LIN {X 0,Y 173.753,Z 484.675,A -85,B 0,C 180,E1 -23523.059,E2 -23523.059} C_VEL
LIN {X 0,Y 169.209,Z 473.205,A -85,B 0,C 180,E1 -23526.461,E2 -23526.461} C_VEL
LIN {X 0,Y 168.375,Z 468.327,A -85,B 0,C 180,E1 -23527.591,E2 -23527.591} C_VEL
LIN {X 0,Y 167.185,Z 457.036,A -85,B 0,C 180,E1 -23529.768,E2 -23529.768} C_VEL
LIN {X 0,Y 165.536,Z 447.869,A -85,B 0,C 180,E1 -23531.391,E2 -23531.391} C_VEL
LIN {X 0,Y 162.65,Z 440.385,A -85,B 0,C 180,E1 -23532.953,E2 -23532.953} C_VEL
LIN {X 0,Y 161.077,Z 436.839,A -85,B 0,C 180,E1 -23533.695,E2 -23533.695} C_VEL
LIN {X 0,Y 159.754,Z 433.864,A -85,B 0,C 180,E1 -23534.312,E2 -23534.312} C_VEL
LIN {X 0,Y 159.528,Z 432.773,A -85,B 0,C 180,E1 -23534.505,E2 -23534.505} C_VEL
LIN {X 0,Y 158.912,Z 429.909,A -85,B 0,C 180,E1 -23538.756,E2 -23538.756} C_VEL
LIN {X 0,Y 158.146,Z 426.115,A -85,B 0,C 180,E1 -23544.709,E2 -23544.709} C_VEL
LIN {X 0,Y 157.921,Z 424.301,A -85,B 0,C 180,E1 -23547.739,E2 -23547.739} C_VEL
LIN {X 0,Y 157.435,Z 421.293,A -85,B 0,C 180,E1 -23553.237,E2 -23553.237} C_VEL
LIN {X 0,Y 157.384,Z 420.882,A -85,B 0,C 180,E1 -23554.19,E2 -23554.19} C_VEL
LIN {X 0,Y 157.405,Z 420.883,A -85,B 0,C 180,E1 -23559.669,E2 -23559.669} C_VEL
LIN {X 0,Y 157.452,Z 420.881,A -85,B 0,C 180,E1 -23564.465,E2 -23564.465} C_VEL
LIN {X 0,Y 157.7,Z 420.846,A -85,B 0,C 180,E1 -23569.731,E2 -23569.731} C_VEL
LIN {X 0,Y 157.777,Z 420.836,A -85,B 0,C 180,E1 -23572.32,E2 -23572.32} C_VEL
LIN {X 0,Y 158.266,Z 420.771,A -85,B 0,C 180,E1 -23580,E2 -23580} C_VEL
LIN {X 0,Y 157.819,Z 420.787,A -85,B 0,C 180,E1 -23587.677,E2 -23587.677} C_VEL
LIN {X 0,Y 157.694,Z 420.835,A -85,B 0,C 180,E1 -23591.319,E2 -23591.319} C_VEL
LIN {X 0,Y 157.488,Z 420.862,A -85,B 0,C 180,E1 -23595.53,E2 -23595.53} C_VEL
LIN {X 0,Y 157.38,Z 420.844,A -85,B 0,C 180,E1 -23600.931,E2 -23600.931} C_VEL
LIN {X 0,Y 157.32,Z 420.888,A -85,B 0,C 180,E1 -23606.679,E2 -23606.679} C_VEL
LIN {X 0,Y 157.284,Z 420.858,A -85,B 0,C 180,E1 -23612.425,E2 -23612.425} C_VEL
LIN {X 0,Y 157.277,Z 420.888,A -85,B 0,C 180,E1 -23616.447,E2 -23616.447} C_VEL
LIN {X 0,Y 157.219,Z 420.881,A -85,B 0,C 180,E1 -23622.108,E2 -23622.108} C_VEL
LIN {X 0,Y 157.218,Z 420.901,A -85,B 0,C 180,E1 -23627.886,E2 -23627.886} C_VEL
LIN {X 0,Y 157.275,Z 420.879,A -85,B 0,C 180,E1 -23633.547,E2 -23633.547} C_VEL
LIN {X 0,Y 157.3,Z 420.889,A -85,B 0,C 180,E1 -23638.092,E2 -23638.092} C_VEL
LIN {X 0,Y 157.329,Z 420.894,A -85,B 0,C 180,E1 -23643.462,E2 -23643.462} C_VEL
LIN {X 0,Y 157.389,Z 421.075,A -85,B 0,C 180,E1 -23648.38,E2 -23648.38} C_VEL
LIN {X 0,Y 158.508,Z 423.935,A -85,B 0,C 180,E1 -23648.983,E2 -23648.983} C_VEL
LIN {X 0,Y 159.904,Z 425.81,A -85,B 0,C 180,E1 -23649.596,E2 -23649.596} C_VEL
LIN {X 0,Y 165.093,Z 435.684,A -85,B 0,C 180,E1 -23652.243,E2 -23652.243} C_VEL
LIN {X 0,Y 168.754,Z 444.416,A -85,B 0,C 180,E1 -23654.504,E2 -23654.504} C_VEL
LIN {X 0,Y 170.95,Z 453.105,A -85,B 0,C 180,E1 -23656.647,E2 -23656.647} C_VEL
LIN {X 0,Y 172.347,Z 463.912,A -85,B 0,C 180,E1 -23659.379,E2 -23659.379} C_VEL
LIN {X 0,Y 172.769,Z 470.682,A -85,B 0,C 180,E1 -23661.268,E2 -23661.268} C_VEL
LIN {X 0,Y 169.378,Z 481.319,A -85,B 0,C 180,E1 -23664.012,E2 -23664.012} C_VEL
LIN {X 0,Y 166.199,Z 490.266,A -85,B 0,C 180,E1 -23666.965,E2 -23666.965} C_VEL
LIN {X 0,Y 163.011,Z 498.684,A -85,B 0,C 180,E1 -23670.539,E2 -23670.539} C_VEL
LIN {X 0,Y 160.315,Z 505.722,A -85,B 0,C 180,E1 -23674.395,E2 -23674.395} C_VEL
LIN {X 0,Y 158.539,Z 510.345,A -85,B 0,C 180,E1 -23677.637,E2 -23677.637} C_VEL
LIN {X 0,Y 156.952,Z 514.644,A -85,B 0,C 180,E1 -23681.489,E2 -23681.489} C_VEL
LIN {X 0,Y 155.686,Z 518.09,A -85,B 0,C 180,E1 -23685.71,E2 -23685.71} C_VEL
LIN {X 0,Y 155.154,Z 519.7,A -85,B 0,C 180,E1 -23688.481,E2 -23688.481} C_VEL
LIN {X 0,Y 154.951,Z 520.827,A -85,B 0,C 180,E1 -23691.27,E2 -23691.27} C_VEL
LIN {X 0,Y 155.024,Z 521.64,A -85,B 0,C 180,E1 -23694.948,E2 -23694.948} C_VEL
LIN {X 0,Y 155.781,Z 521.51,A -85,B 0,C 180,E1 -23699.746,E2 -23699.746} C_VEL
LIN {X 0,Y 156.591,Z 520.823,A -85,B 0,C 180,E1 -23702.58,E2 -23702.58} C_VEL
LIN {X 0,Y 158.428,Z 518.701,A -85,B 0,C 180,E1 -23707.014,E2 -23707.014} C_VEL
LIN {X 0,Y 160.723,Z 515.657,A -85,B 0,C 180,E1 -23710.981,E2 -23710.981} C_VEL
LIN {X 0,Y 163.815,Z 511.176,A -85,B 0,C 180,E1 -23715.055,E2 -23715.055} C_VEL
LIN {X 0,Y 167.633,Z 505.239,A -85,B 0,C 180,E1 -23718.986,E2 -23718.986} C_VEL
LIN {X 0,Y 171.512,Z 498.72,A -85,B 0,C 180,E1 -23722.247,E2 -23722.247} C_VEL
LIN {X 0,Y 175.508,Z 491.246,A -85,B 0,C 180,E1 -23725.165,E2 -23725.165} C_VEL
LIN {X 0,Y 180.132,Z 481.611,A -85,B 0,C 180,E1 -23728.049,E2 -23728.049} C_VEL
LIN {X 0,Y 180.912,Z 479.34,A -85,B 0,C 180,E1 -23728.711,E2 -23728.711} C_VEL
LIN {X 0,Y 180.836,Z 471.499,A -85,B 0,C 180,E1 -23731.57,E2 -23731.57} C_VEL
LIN {X 0,Y 180.166,Z 465.408,A -85,B 0,C 180,E1 -23733.78,E2 -23733.78} C_VEL
LIN {X 0,Y 178.357,Z 457.69,A -85,B 0,C 180,E1 -23736.794,E2 -23736.794} C_VEL
LIN {X 0,Y 175.967,Z 451.426,A -85,B 0,C 180,E1 -23739.545,E2 -23739.545} C_VEL
LIN {X 0,Y 174.463,Z 447.925,A -85,B 0,C 180,E1 -23741.2,E2 -23741.2} C_VEL
LIN {X 0,Y 171.091,Z 441.961,A -85,B 0,C 180,E1 -23744.514,E2 -23744.514} C_VEL
LIN {X 0,Y 168.78,Z 438.136,A -85,B 0,C 180,E1 -23746.914,E2 -23746.914} C_VEL
LIN {X 0,Y 166.844,Z 434.787,A -85,B 0,C 180,E1 -23749.072,E2 -23749.072} C_VEL
LIN {X 0,Y 166.071,Z 433.805,A -85,B 0,C 180,E1 -23749.902,E2 -23749.902} C_VEL
LIN {X 0,Y 163.624,Z 430.698,A -85,B 0,C 180,E1 -23752.752,E2 -23752.752} C_VEL
LIN {X 0,Y 162.937,Z 429.155,A -85,B 0,C 180,E1 -23753.811,E2 -23753.811} C_VEL
LIN {X 0,Y 160.283,Z 427.137,A -85,B 0,C 180,E1 -23757.33,E2 -23757.33} C_VEL
LIN {X 0,Y 159.035,Z 424.704,A -85,B 0,C 180,E1 -23759.842,E2 -23759.842} C_VEL
LIN {X 0,Y 158.704,Z 423.885,A -85,B 0,C 180,E1 -23760.793,E2 -23760.793} C_VEL
LIN {X 0,Y 158.42,Z 424.419,A -85,B 0,C 180,E1 -23767.648,E2 -23767.648} C_VEL
LIN {X 0,Y 158.386,Z 425.205,A -85,B 0,C 180,E1 -23772.819,E2 -23772.819} C_VEL
LIN {X 0,Y 158.473,Z 426.363,A -85,B 0,C 180,E1 -23778.086,E2 -23778.086} C_VEL
LIN {X 0,Y 158.651,Z 427.629,A -85,B 0,C 180,E1 -23782.159,E2 -23782.159} C_VEL
LIN {X 0,Y 159.752,Z 430.657,A -85,B 0,C 180,E1 -23784.531,E2 -23784.531} C_VEL
LIN {X 0,Y 163.129,Z 435.032,A -85,B 0,C 180,E1 -23789.168,E2 -23789.168} C_VEL
LIN {X 0,Y 163.642,Z 435.727,A -85,B 0,C 180,E1 -23789.774,E2 -23789.774} C_VEL
LIN {X 0,Y 165.237,Z 439.58,A -85,B 0,C 180,E1 -23791.945,E2 -23791.945} C_VEL
LIN {X 0,Y 167.427,Z 442.4,A -85,B 0,C 180,E1 -23794.092,E2 -23794.092} C_VEL
LIN {X 0,Y 169.032,Z 446.242,A -85,B 0,C 180,E1 -23795.965,E2 -23795.965} C_VEL
LIN {X 0,Y 170.595,Z 448.842,A -85,B 0,C 180,E1 -23797.421,E2 -23797.421} C_VEL
LIN {X 0,Y 172.933,Z 453.744,A -85,B 0,C 180,E1 -23799.723,E2 -23799.723} C_VEL
LIN {X 0,Y 176.427,Z 462.831,A -85,B 0,C 180,E1 -23803.407,E2 -23803.407} C_VEL
LIN {X 0,Y 177.631,Z 467.087,A -85,B 0,C 180,E1 -23804.92,E2 -23804.92} C_VEL
LIN {X 0,Y 178.101,Z 473.747,A -85,B 0,C 180,E1 -23806.829,E2 -23806.829} C_VEL
LIN {X 0,Y 177.816,Z 483.644,A -85,B 0,C 180,E1 -23809.587,E2 -23809.587} C_VEL
LIN {X 0,Y 176.545,Z 493.509,A -85,B 0,C 180,E1 -23812.489,E2 -23812.489} C_VEL
LIN {X 0,Y 174.717,Z 501.481,A -85,B 0,C 180,E1 -23815.041,E2 -23815.041} C_VEL
LIN {X 0,Y 172.499,Z 508.067,A -85,B 0,C 180,E1 -23817.334,E2 -23817.334} C_VEL
LIN {X 0,Y 168.012,Z 516.355,A -85,B 0,C 180,E1 -23820.566,E2 -23820.566} C_VEL
LIN {X 0,Y 164.25,Z 523.057,A -85,B 0,C 180,E1 -23823.97,E2 -23823.97} C_VEL
LIN {X 0,Y 161.64,Z 527.705,A -85,B 0,C 180,E1 -23826.969,E2 -23826.969} C_VEL
LIN {X 0,Y 158.969,Z 532.18,A -85,B 0,C 180,E1 -23830.641,E2 -23830.641} C_VEL
LIN {X 0,Y 156.937,Z 535.616,A -85,B 0,C 180,E1 -23834.419,E2 -23834.419} C_VEL
LIN {X 0,Y 155.458,Z 538.718,A -85,B 0,C 180,E1 -23839.587,E2 -23839.587} C_VEL
LIN {X 0,Y 155.109,Z 539.685,A -85,B 0,C 180,E1 -23842.193,E2 -23842.193} C_VEL
LIN {X 0,Y 154.991,Z 540.343,A -85,B 0,C 180,E1 -23846.019,E2 -23846.019} C_VEL
LIN {X 0,Y 155.28,Z 540.125,A -85,B 0,C 180,E1 -23850.005,E2 -23850.005} C_VEL
LIN {X 0,Y 155.086,Z 538.698,A -85,B 0,C 180,E1 -23854.455,E2 -23854.455} C_VEL
LIN {X 0,Y 155.202,Z 536.785,A -85,B 0,C 180,E1 -23857.813,E2 -23857.813} C_VEL
LIN {X 0,Y 155.82,Z 533.633,A -85,B 0,C 180,E1 -23861.715,E2 -23861.715} C_VEL
LIN {X 0,Y 156.959,Z 529.391,A -85,B 0,C 180,E1 -23865.589,E2 -23865.589} C_VEL
LIN {X 0,Y 159.262,Z 522.952,A -85,B 0,C 180,E1 -23870.003,E2 -23870.003} C_VEL
LIN {X 0,Y 161.829,Z 515.818,A -85,B 0,C 180,E1 -23873.726,E2 -23873.726} C_VEL
LIN {X 0,Y 165.001,Z 507.05,A -85,B 0,C 180,E1 -23877.255,E2 -23877.255} C_VEL
LIN {X 0,Y 167.404,Z 499.95,A -85,B 0,C 180,E1 -23879.562,E2 -23879.562} C_VEL
LIN {X 0,Y 168.435,Z 489.968,A -85,B 0,C 180,E1 -23882.499,E2 -23882.499} C_VEL
LIN {X 0,Y 168.701,Z 478.718,A -85,B 0,C 180,E1 -23885.342,E2 -23885.342} C_VEL
LIN {X 0,Y 168.375,Z 468.327,A -85,B 0,C 180,E1 -23887.591,E2 -23887.591} C_VEL
LIN {X 0,Y 167.531,Z 463.422,A -85,B 0,C 180,E1 -23888.683,E2 -23888.683} C_VEL
LIN {X 0,Y 165.736,Z 458.883,A -85,B 0,C 180,E1 -23889.856,E2 -23889.856} C_VEL
LIN {X 0,Y 160.747,Z 450.349,A -85,B 0,C 180,E1 -23892.302,E2 -23892.302} C_VEL
LIN {X 0,Y 157.439,Z 444.408,A -85,B 0,C 180,E1 -23893.892,E2 -23893.892} C_VEL
LIN {X 0,Y 154.137,Z 436.914,A -85,B 0,C 180,E1 -23895.641,E2 -23895.641} C_VEL
LIN {X 0,Y 152.568,Z 433.873,A -85,B 0,C 180,E1 -23896.41,E2 -23896.41} C_VEL
LIN {X 0,Y 152.182,Z 432.293,A -85,B 0,C 180,E1 -23896.743,E2 -23896.743} C_VEL
LIN {X 0,Y 151.359,Z 428.42,A -85,B 0,C 180,E1 -23902.87,E2 -23902.87} C_VEL
LIN {X 0,Y 150.793,Z 424.852,A -85,B 0,C 180,E1 -23909.157,E2 -23909.157} C_VEL
LIN {X 0,Y 150.334,Z 421.76,A -85,B 0,C 180,E1 -23915.302,E2 -23915.302} C_VEL
LIN {X 0,Y 150.371,Z 421.761,A -85,B 0,C 180,E1 -23920.903,E2 -23920.903} C_VEL
LIN {X 0,Y 150.441,Z 421.754,A -85,B 0,C 180,E1 -23926.492,E2 -23926.492} C_VEL
LIN {X 0,Y 150.622,Z 421.728,A -85,B 0,C 180,E1 -23929.243,E2 -23929.243} C_VEL
LIN {X 0,Y 150.715,Z 421.715,A -85,B 0,C 180,E1 -23931.958,E2 -23931.958} C_VEL
LIN {X 0,Y 151.226,Z 421.648,A -85,B 0,C 180,E1 -23940,E2 -23940} C_VEL
LIN {X 0,Y 150.754,Z 421.667,A -85,B 0,C 180,E1 -23948.039,E2 -23948.039} C_VEL
LIN {X 0,Y 150.625,Z 421.716,A -85,B 0,C 180,E1 -23951.505,E2 -23951.505} C_VEL
LIN {X 0,Y 150.393,Z 421.741,A -85,B 0,C 180,E1 -23956.283,E2 -23956.283} C_VEL
LIN {X 0,Y 150.361,Z 421.716,A -85,B 0,C 180,E1 -23960.79,E2 -23960.79} C_VEL
LIN {X 0,Y 150.251,Z 421.77,A -85,B 0,C 180,E1 -23967.278,E2 -23967.278} C_VEL
LIN {X 0,Y 150.223,Z 421.736,A -85,B 0,C 180,E1 -23972.629,E2 -23972.629} C_VEL
LIN {X 0,Y 150.186,Z 421.775,A -85,B 0,C 180,E1 -23977.469,E2 -23977.469} C_VEL
LIN {X 0,Y 150.158,Z 421.766,A -85,B 0,C 180,E1 -23981.502,E2 -23981.502} C_VEL
LIN {X 0,Y 150.133,Z 421.764,A -85,B 0,C 180,E1 -23985.392,E2 -23985.392} C_VEL
LIN {X 0,Y 150.158,Z 421.78,A -85,B 0,C 180,E1 -23989.055,E2 -23989.055} C_VEL
LIN {X 0,Y 150.186,Z 421.758,A -85,B 0,C 180,E1 -23992.704,E2 -23992.704} C_VEL
LIN {X 0,Y 150.222,Z 421.775,A -85,B 0,C 180,E1 -23997.364,E2 -23997.364} C_VEL
LIN {X 0,Y 150.251,Z 421.776,A -85,B 0,C 180,E1 -24002.713,E2 -24002.713} C_VEL
LIN {X 0,Y 150.284,Z 421.83,A -85,B 0,C 180,E1 -24006.221,E2 -24006.221} C_VEL
LIN {X 0,Y 151.27,Z 424.573,A -85,B 0,C 180,E1 -24006.829,E2 -24006.829} C_VEL
LIN {X 0,Y 152.832,Z 426.794,A -85,B 0,C 180,E1 -24007.597,E2 -24007.597} C_VEL
LIN {X 0,Y 154.829,Z 430.108,A -85,B 0,C 180,E1 -24008.615,E2 -24008.615} C_VEL
LIN {X 0,Y 160.094,Z 440.601,A -85,B 0,C 180,E1 -24011.69,E2 -24011.69} C_VEL
LIN {X 0,Y 163.298,Z 449.135,A -85,B 0,C 180,E1 -24014.079,E2 -24014.079} C_VEL
LIN {X 0,Y 164.823,Z 455.727,A -85,B 0,C 180,E1 -24015.821,E2 -24015.821} C_VEL
LIN {X 0,Y 166.061,Z 467.475,A -85,B 0,C 180,E1 -24019.048,E2 -24019.048} C_VEL
LIN {X 0,Y 166.289,Z 471.524,A -85,B 0,C 180,E1 -24020.263,E2 -24020.263} C_VEL
LIN {X 0,Y 162.824,Z 482.07,A -85,B 0,C 180,E1 -24023.098,E2 -24023.098} C_VEL
LIN {X 0,Y 159.462,Z 491.064,A -85,B 0,C 180,E1 -24026.205,E2 -24026.205} C_VEL
LIN {X 0,Y 156.081,Z 499.578,A -85,B 0,C 180,E1 -24029.995,E2 -24029.995} C_VEL
LIN {X 0,Y 153.342,Z 506.408,A -85,B 0,C 180,E1 -24033.937,E2 -24033.937} C_VEL
LIN {X 0,Y 151.177,Z 511.81,A -85,B 0,C 180,E1 -24038.012,E2 -24038.012} C_VEL
LIN {X 0,Y 149.56,Z 515.99,A -85,B 0,C 180,E1 -24042.202,E2 -24042.202} C_VEL
LIN {X 0,Y 148.413,Z 519.07,A -85,B 0,C 180,E1 -24046.501,E2 -24046.501} C_VEL
LIN {X 0,Y 147.979,Z 520.528,A -85,B 0,C 180,E1 -24049.412,E2 -24049.412} C_VEL
LIN {X 0,Y 147.827,Z 521.555,A -85,B 0,C 180,E1 -24052.348,E2 -24052.348} C_VEL
LIN {X 0,Y 147.975,Z 522.1,A -85,B 0,C 180,E1 -24055.525,E2 -24055.525} C_VEL
LIN {X 0,Y 148.359,Z 522.166,A -85,B 0,C 180,E1 -24058.269,E2 -24058.269} C_VEL
LIN {X 0,Y 149.353,Z 521.577,A -85,B 0,C 180,E1 -24062.112,E2 -24062.112} C_VEL
LIN {X 0,Y 151.319,Z 519.586,A -85,B 0,C 180,E1 -24067.134,E2 -24067.134} C_VEL
LIN {X 0,Y 153.807,Z 516.595,A -85,B 0,C 180,E1 -24071.487,E2 -24071.487} C_VEL
LIN {X 0,Y 157.041,Z 512.303,A -85,B 0,C 180,E1 -24075.72,E2 -24075.72} C_VEL
LIN {X 0,Y 161.031,Z 506.509,A -85,B 0,C 180,E1 -24079.818,E2 -24079.818} C_VEL
LIN {X 0,Y 165.708,Z 499.132,A -85,B 0,C 180,E1 -24083.68,E2 -24083.68} C_VEL
LIN {X 0,Y 169.998,Z 491.579,A -85,B 0,C 180,E1 -24086.686,E2 -24086.686} C_VEL
LIN {X 0,Y 174.948,Z 481.709,A -85,B 0,C 180,E1 -24089.69,E2 -24089.69} C_VEL
LIN {X 0,Y 175.119,Z 474.619,A -85,B 0,C 180,E1 -24092.476,E2 -24092.476} C_VEL
LIN {X 0,Y 174.394,Z 466.778,A -85,B 0,C 180,E1 -24095.602,E2 -24095.602} C_VEL
LIN {X 0,Y 172.779,Z 460.047,A -85,B 0,C 180,E1 -24098.526,E2 -24098.526} C_VEL
LIN {X 0,Y 170.226,Z 453.171,A -85,B 0,C 180,E1 -24101.961,E2 -24101.961} C_VEL
LIN {X 0,Y 166.794,Z 446.29,A -85,B 0,C 180,E1 -24106.041,E2 -24106.041} C_VEL
LIN {X 0,Y 163.603,Z 440.467,A -85,B 0,C 180,E1 -24110.106,E2 -24110.106} C_VEL
LIN {X 0,Y 161.169,Z 437.172,A -85,B 0,C 180,E1 -24113.31,E2 -24113.31} C_VEL
LIN {X 0,Y 160.584,Z 435.793,A -85,B 0,C 180,E1 -24114.356,E2 -24114.356} C_VEL
LIN {X 0,Y 158.165,Z 433.6,A -85,B 0,C 180,E1 -24118.09,E2 -24118.09} C_VEL
LIN {X 0,Y 157.097,Z 430.867,A -85,B 0,C 180,E1 -24120.961,E2 -24120.961} C_VEL
LIN {X 0,Y 154.798,Z 430.545,A -85,B 0,C 180,E1 -24127.828,E2 -24127.828} C_VEL
LIN {X 0,Y 154.562,Z 431.276,A -85,B 0,C 180,E1 -24133.141,E2 -24133.141} C_VEL
LIN {X 0,Y 156.749,Z 434.093,A -85,B 0,C 180,E1 -24141.208,E2 -24141.208} C_VEL
LIN {X 0,Y 158.112,Z 437.966,A -85,B 0,C 180,E1 -24144.628,E2 -24144.628} C_VEL
LIN {X 0,Y 160.988,Z 442.005,A -85,B 0,C 180,E1 -24148.94,E2 -24148.94} C_VEL
LIN {X 0,Y 162.573,Z 446.035,A -85,B 0,C 180,E1 -24151.438,E2 -24151.438} C_VEL
LIN {X 0,Y 163.813,Z 447.698,A -85,B 0,C 180,E1 -24152.812,E2 -24152.812} C_VEL
LIN {X 0,Y 166.556,Z 453.649,A -85,B 0,C 180,E1 -24156.21,E2 -24156.21} C_VEL
LIN {X 0,Y 169.063,Z 459.815,A -85,B 0,C 180,E1 -24159.236,E2 -24159.236} C_VEL
LIN {X 0,Y 171.629,Z 467.332,A -85,B 0,C 180,E1 -24162.525,E2 -24162.525} C_VEL
LIN {X 0,Y 172.625,Z 472.125,A -85,B 0,C 180,E1 -24164.297,E2 -24164.297} C_VEL
LIN {X 0,Y 172.583,Z 480.365,A -85,B 0,C 180,E1 -24166.786,E2 -24166.786} C_VEL
LIN {X 0,Y 171.457,Z 490.287,A -85,B 0,C 180,E1 -24169.798,E2 -24169.798} C_VEL
LIN {X 0,Y 169.619,Z 499.083,A -85,B 0,C 180,E1 -24172.676,E2 -24172.676} C_VEL
LIN {X 0,Y 167.17,Z 506.719,A -85,B 0,C 180,E1 -24175.427,E2 -24175.427} C_VEL
LIN {X 0,Y 164.15,Z 512.526,A -85,B 0,C 180,E1 -24177.65,E2 -24177.65} C_VEL
LIN {X 0,Y 159.751,Z 519.896,A -85,B 0,C 180,E1 -24181.064,E2 -24181.064} C_VEL
LIN {X 0,Y 156.249,Z 525.875,A -85,B 0,C 180,E1 -24184.709,E2 -24184.709} C_VEL
LIN {X 0,Y 153.122,Z 530.645,A -85,B 0,C 180,E1 -24188.464,E2 -24188.464} C_VEL
LIN {X 0,Y 150.724,Z 534.341,A -85,B 0,C 180,E1 -24192.363,E2 -24192.363} C_VEL
LIN {X 0,Y 149.115,Z 537.064,A -85,B 0,C 180,E1 -24196.375,E2 -24196.375} C_VEL
LIN {X 0,Y 148.463,Z 538.386,A -85,B 0,C 180,E1 -24199.09,E2 -24199.09} C_VEL
LIN {X 0,Y 148.042,Z 539.306,A -85,B 0,C 180,E1 -24201.818,E2 -24201.818} C_VEL
LIN {X 0,Y 147.915,Z 539.947,A -85,B 0,C 180,E1 -24206.193,E2 -24206.193} C_VEL
LIN {X 0,Y 148.192,Z 539.65,A -85,B 0,C 180,E1 -24210.005,E2 -24210.005} C_VEL
LIN {X 0,Y 147.996,Z 538.335,A -85,B 0,C 180,E1 -24214.251,E2 -24214.251} C_VEL
LIN {X 0,Y 148.309,Z 535.251,A -85,B 0,C 180,E1 -24219.552,E2 -24219.552} C_VEL
LIN {X 0,Y 149.173,Z 531.684,A -85,B 0,C 180,E1 -24223.63,E2 -24223.63} C_VEL
LIN {X 0,Y 150.752,Z 526.998,A -85,B 0,C 180,E1 -24227.645,E2 -24227.645} C_VEL
LIN {X 0,Y 153.39,Z 519.918,A -85,B 0,C 180,E1 -24232.215,E2 -24232.215} C_VEL
LIN {X 0,Y 156.109,Z 512.72,A -85,B 0,C 180,E1 -24235.789,E2 -24235.789} C_VEL
LIN {X 0,Y 159.296,Z 504.366,A -85,B 0,C 180,E1 -24239.038,E2 -24239.038} C_VEL
LIN {X 0,Y 160.802,Z 499.788,A -85,B 0,C 180,E1 -24240.541,E2 -24240.541} C_VEL
LIN {X 0,Y 161.84,Z 489.809,A -85,B 0,C 180,E1 -24243.625,E2 -24243.625} C_VEL
LIN {X 0,Y 162.213,Z 480.188,A -85,B 0,C 180,E1 -24246.183,E2 -24246.183} C_VEL
LIN {X 0,Y 162.028,Z 469.456,A -85,B 0,C 180,E1 -24248.67,E2 -24248.67} C_VEL
LIN {X 0,Y 160.969,Z 457.998,A -85,B 0,C 180,E1 -24251.042,E2 -24251.042} C_VEL
LIN {X 0,Y 159.68,Z 450.554,A -85,B 0,C 180,E1 -24252.504,E2 -24252.504} C_VEL
LIN {X 0,Y 157.439,Z 444.408,A -85,B 0,C 180,E1 -24253.892,E2 -24253.892} C_VEL
LIN {X 0,Y 155.429,Z 441.819,A -85,B 0,C 180,E1 -24254.754,E2 -24254.754} C_VEL
LIN {X 0,Y 146.78,Z 436.045,A -85,B 0,C 180,E1 -24258.088,E2 -24258.088} C_VEL
LIN {X 0,Y 145.32,Z 433.745,A -85,B 0,C 180,E1 -24258.807,E2 -24258.807} C_VEL
LIN {X 0,Y 145.124,Z 433.196,A -85,B 0,C 180,E1 -24258.926,E2 -24258.926} C_VEL
LIN {X 0,Y 144.775,Z 431.726,A -85,B 0,C 180,E1 -24259.226,E2 -24259.226} C_VEL
LIN {X 0,Y 144.051,Z 427.842,A -85,B 0,C 180,E1 -24266.045,E2 -24266.045} C_VEL
LIN {X 0,Y 143.584,Z 424.839,A -85,B 0,C 180,E1 -24271.778,E2 -24271.778} C_VEL
LIN {X 0,Y 143.246,Z 422.643,A -85,B 0,C 180,E1 -24276.507,E2 -24276.507} C_VEL
LIN {X 0,Y 143.318,Z 422.639,A -85,B 0,C 180,E1 -24279.924,E2 -24279.924} C_VEL
LIN {X 0,Y 143.364,Z 422.634,A -85,B 0,C 180,E1 -24285.811,E2 -24285.811} C_VEL
LIN {X 0,Y 143.548,Z 422.611,A -85,B 0,C 180,E1 -24288.706,E2 -24288.706} C_VEL
LIN {X 0,Y 143.636,Z 422.597,A -85,B 0,C 180,E1 -24291.559,E2 -24291.559} C_VEL
LIN {X 0,Y 144.185,Z 422.525,A -85,B 0,C 180,E1 -24300,E2 -24300} C_VEL
LIN {X 0,Y 143.675,Z 422.55,A -85,B 0,C 180,E1 -24308.438,E2 -24308.438} C_VEL
LIN {X 0,Y 143.559,Z 422.597,A -85,B 0,C 180,E1 -24311.711,E2 -24311.711} C_VEL
LIN {X 0,Y 143.327,Z 422.611,A -85,B 0,C 180,E1 -24317.11,E2 -24317.11} C_VEL
LIN {X 0,Y 143.287,Z 422.598,A -85,B 0,C 180,E1 -24321.252,E2 -24321.252} C_VEL
LIN {X 0,Y 143.198,Z 422.645,A -85,B 0,C 180,E1 -24327.933,E2 -24327.933} C_VEL
LIN {X 0,Y 143.152,Z 422.617,A -85,B 0,C 180,E1 -24333.417,E2 -24333.417} C_VEL
LIN {X 0,Y 143.071,Z 422.661,A -85,B 0,C 180,E1 -24339.687,E2 -24339.687} C_VEL
LIN {X 0,Y 143.045,Z 422.638,A -85,B 0,C 180,E1 -24343.459,E2 -24343.459} C_VEL
LIN {X 0,Y 143.073,Z 422.661,A -85,B 0,C 180,E1 -24347.462,E2 -24347.462} C_VEL
LIN {X 0,Y 143.084,Z 422.643,A -85,B 0,C 180,E1 -24351.803,E2 -24351.803} C_VEL
LIN {X 0,Y 143.189,Z 422.651,A -85,B 0,C 180,E1 -24357.317,E2 -24357.317} C_VEL
LIN {X 0,Y 143.189,Z 422.655,A -85,B 0,C 180,E1 -24363.78,E2 -24363.78} C_VEL
LIN {X 0,Y 144.206,Z 425.52,A -85,B 0,C 180,E1 -24364.488,E2 -24364.488} C_VEL
LIN {X 0,Y 145.853,Z 427.689,A -85,B 0,C 180,E1 -24365.372,E2 -24365.372} C_VEL
LIN {X 0,Y 151.079,Z 437.022,A -85,B 0,C 180,E1 -24368.493,E2 -24368.493} C_VEL
LIN {X 0,Y 155.548,Z 446.838,A -85,B 0,C 180,E1 -24371.591,E2 -24371.591} C_VEL
LIN {X 0,Y 157.903,Z 454.279,A -85,B 0,C 180,E1 -24373.823,E2 -24373.823} C_VEL
LIN {X 0,Y 158.998,Z 461.758,A -85,B 0,C 180,E1 -24375.926,E2 -24375.926} C_VEL
LIN {X 0,Y 159.708,Z 470.646,A -85,B 0,C 180,E1 -24378.606,E2 -24378.606} C_VEL
LIN {X 0,Y 159.792,Z 472.598,A -85,B 0,C 180,E1 -24379.238,E2 -24379.238} C_VEL
LIN {X 0,Y 156.871,Z 481.215,A -85,B 0,C 180,E1 -24381.623,E2 -24381.623} C_VEL
LIN {X 0,Y 153.398,Z 490.265,A -85,B 0,C 180,E1 -24384.738,E2 -24384.738} C_VEL
LIN {X 0,Y 150.358,Z 497.708,A -85,B 0,C 180,E1 -24387.986,E2 -24387.986} C_VEL
LIN {X 0,Y 147.639,Z 504.135,A -85,B 0,C 180,E1 -24391.512,E2 -24391.512} C_VEL
LIN {X 0,Y 145.187,Z 509.901,A -85,B 0,C 180,E1 -24395.55,E2 -24395.55} C_VEL
LIN {X 0,Y 142.994,Z 515.26,A -85,B 0,C 180,E1 -24400.587,E2 -24400.587} C_VEL
LIN {X 0,Y 141.799,Z 518.208,A -85,B 0,C 180,E1 -24404.342,E2 -24404.342} C_VEL
LIN {X 0,Y 140.962,Z 520.627,A -85,B 0,C 180,E1 -24408.686,E2 -24408.686} C_VEL
LIN {X 0,Y 140.761,Z 522.186,A -85,B 0,C 180,E1 -24413.536,E2 -24413.536} C_VEL
LIN {X 0,Y 141.004,Z 522.598,A -85,B 0,C 180,E1 -24416.646,E2 -24416.646} C_VEL
LIN {X 0,Y 141.577,Z 522.563,A -85,B 0,C 180,E1 -24419.756,E2 -24419.756} C_VEL
LIN {X 0,Y 142.497,Z 521.976,A -85,B 0,C 180,E1 -24423.024,E2 -24423.024} C_VEL
LIN {X 0,Y 143.586,Z 521.025,A -85,B 0,C 180,E1 -24425.962,E2 -24425.962} C_VEL
LIN {X 0,Y 145.2,Z 519.384,A -85,B 0,C 180,E1 -24429.247,E2 -24429.247} C_VEL
LIN {X 0,Y 147.965,Z 516.26,A -85,B 0,C 180,E1 -24433.52,E2 -24433.52} C_VEL
LIN {X 0,Y 151.566,Z 511.701,A -85,B 0,C 180,E1 -24437.885,E2 -24437.885} C_VEL
LIN {X 0,Y 156.011,Z 505.695,A -85,B 0,C 180,E1 -24442.021,E2 -24442.021} C_VEL
LIN {X 0,Y 161.103,Z 497.863,A -85,B 0,C 180,E1 -24445.972,E2 -24445.972} C_VEL
LIN {X 0,Y 165.886,Z 489.7,A -85,B 0,C 180,E1 -24449.068,E2 -24449.068} C_VEL
LIN {X 0,Y 169.002,Z 483.889,A -85,B 0,C 180,E1 -24450.832,E2 -24450.832} C_VEL
LIN {X 0,Y 169.424,Z 477.503,A -85,B 0,C 180,E1 -24453.517,E2 -24453.517} C_VEL
LIN {X 0,Y 169.169,Z 471.632,A -85,B 0,C 180,E1 -24456.046,E2 -24456.046} C_VEL
LIN {X 0,Y 167.972,Z 464.902,A -85,B 0,C 180,E1 -24459.167,E2 -24459.167} C_VEL
LIN {X 0,Y 165.835,Z 458.262,A -85,B 0,C 180,E1 -24462.743,E2 -24462.743} C_VEL
LIN {X 0,Y 163.34,Z 452.656,A -85,B 0,C 180,E1 -24466.311,E2 -24466.311} C_VEL
LIN {X 0,Y 160.141,Z 446.233,A -85,B 0,C 180,E1 -24471.164,E2 -24471.164} C_VEL
LIN {X 0,Y 158.515,Z 443.876,A -85,B 0,C 180,E1 -24473.636,E2 -24473.636} C_VEL
LIN {X 0,Y 157.95,Z 442.293,A -85,B 0,C 180,E1 -24474.895,E2 -24474.895} C_VEL
LIN {X 0,Y 156.433,Z 440.982,A -85,B 0,C 180,E1 -24477.425,E2 -24477.425} C_VEL
LIN {X 0,Y 155.059,Z 437.806,A -85,B 0,C 180,E1 -24481.299,E2 -24481.299} C_VEL
LIN {X 0,Y 152.914,Z 437.537,A -85,B 0,C 180,E1 -24489.257,E2 -24489.257} C_VEL
LIN {X 0,Y 153.09,Z 438.741,A -85,B 0,C 180,E1 -24495.137,E2 -24495.137} C_VEL
LIN {X 0,Y 154.688,Z 440.97,A -85,B 0,C 180,E1 -24500.791,E2 -24500.791} C_VEL
LIN {X 0,Y 155.719,Z 444.389,A -85,B 0,C 180,E1 -24503.966,E2 -24503.966} C_VEL
LIN {X 0,Y 157.937,Z 447.777,A -85,B 0,C 180,E1 -24507.855,E2 -24507.855} C_VEL
LIN {X 0,Y 159.304,Z 451.768,A -85,B 0,C 180,E1 -24510.488,E2 -24510.488} C_VEL
LIN {X 0,Y 160.658,Z 454.19,A -85,B 0,C 180,E1 -24512.404,E2 -24512.404} C_VEL
LIN {X 0,Y 163.188,Z 460.792,A -85,B 0,C 180,E1 -24516.235,E2 -24516.235} C_VEL
LIN {X 0,Y 165.458,Z 467.333,A -85,B 0,C 180,E1 -24519.579,E2 -24519.579} C_VEL
LIN {X 0,Y 167.088,Z 473.304,A -85,B 0,C 180,E1 -24522.298,E2 -24522.298} C_VEL
LIN {X 0,Y 167.396,Z 477.452,A -85,B 0,C 180,E1 -24523.812,E2 -24523.812} C_VEL
LIN {X 0,Y 166.698,Z 485.785,A -85,B 0,C 180,E1 -24526.486,E2 -24526.486} C_VEL
LIN {X 0,Y 165.033,Z 494.869,A -85,B 0,C 180,E1 -24529.509,E2 -24529.509} C_VEL
LIN {X 0,Y 162.456,Z 503.778,A -85,B 0,C 180,E1 -24532.731,E2 -24532.731} C_VEL
LIN {X 0,Y 160.638,Z 508.439,A -85,B 0,C 180,E1 -24534.578,E2 -24534.578} C_VEL
LIN {X 0,Y 155.772,Z 516.494,A -85,B 0,C 180,E1 -24537.992,E2 -24537.992} C_VEL
LIN {X 0,Y 152.189,Z 522.016,A -85,B 0,C 180,E1 -24541.003,E2 -24541.003} C_VEL
LIN {X 0,Y 148.657,Z 527.47,A -85,B 0,C 180,E1 -24544.825,E2 -24544.825} C_VEL
LIN {X 0,Y 145.59,Z 531.788,A -85,B 0,C 180,E1 -24548.78,E2 -24548.78} C_VEL
LIN {X 0,Y 143.23,Z 535.088,A -85,B 0,C 180,E1 -24552.884,E2 -24552.884} C_VEL
LIN {X 0,Y 141.454,Z 538.057,A -85,B 0,C 180,E1 -24558.543,E2 -24558.543} C_VEL
LIN {X 0,Y 140.842,Z 539.387,A -85,B 0,C 180,E1 -24564.278,E2 -24564.278} C_VEL
LIN {X 0,Y 140.864,Z 539.471,A -85,B 0,C 180,E1 -24567.146,E2 -24567.146} C_VEL
LIN {X 0,Y 141.105,Z 539.171,A -85,B 0,C 180,E1 -24570.005,E2 -24570.005} C_VEL
LIN {X 0,Y 140.925,Z 537.929,A -85,B 0,C 180,E1 -24574.117,E2 -24574.117} C_VEL
LIN {X 0,Y 141.3,Z 534.615,A -85,B 0,C 180,E1 -24580.031,E2 -24580.031} C_VEL
LIN {X 0,Y 142.24,Z 530.977,A -85,B 0,C 180,E1 -24584.308,E2 -24584.308} C_VEL
LIN {X 0,Y 143.959,Z 526.217,A -85,B 0,C 180,E1 -24588.507,E2 -24588.507} C_VEL
LIN {X 0,Y 146.823,Z 519.058,A -85,B 0,C 180,E1 -24593.265,E2 -24593.265} C_VEL
LIN {X 0,Y 149.962,Z 511.09,A -85,B 0,C 180,E1 -24597.264,E2 -24597.264} C_VEL
LIN {X 0,Y 153.745,Z 501.447,A -85,B 0,C 180,E1 -24600.953,E2 -24600.953} C_VEL
LIN {X 0,Y 155.112,Z 492.417,A -85,B 0,C 180,E1 -24603.972,E2 -24603.972} C_VEL
LIN {X 0,Y 155.741,Z 481.499,A -85,B 0,C 180,E1 -24607.131,E2 -24607.131} C_VEL
LIN {X 0,Y 155.736,Z 470.304,A -85,B 0,C 180,E1 -24609.899,E2 -24609.899} C_VEL
LIN {X 0,Y 154.87,Z 459.374,A -85,B 0,C 180,E1 -24612.319,E2 -24612.319} C_VEL
LIN {X 0,Y 153.942,Z 453.583,A -85,B 0,C 180,E1 -24613.551,E2 -24613.551} C_VEL
LIN {X 0,Y 150.558,Z 444.438,A -85,B 0,C 180,E1 -24615.869,E2 -24615.869} C_VEL
LIN {X 0,Y 146.799,Z 436.365,A -85,B 0,C 180,E1 -24618.029,E2 -24618.029} C_VEL
LIN {X 0,Y 145.124,Z 433.196,A -85,B 0,C 180,E1 -24618.926,E2 -24618.926} C_VEL
LIN {X 0,Y 144.246,Z 431.755,A -85,B 0,C 180,E1 -24619.567,E2 -24619.567} C_VEL
LIN {X 0,Y 139.809,Z 429.739,A -85,B 0,C 180,E1 -24623.988,E2 -24623.988} C_VEL
LIN {X 0,Y 137.652,Z 428.46,A -85,B 0,C 180,E1 -24627.481,E2 -24627.481} C_VEL
LIN {X 0,Y 136.644,Z 426.536,A -85,B 0,C 180,E1 -24631.067,E2 -24631.067} C_VEL
LIN {X 0,Y 136.268,Z 423.809,A -85,B 0,C 180,E1 -24637.116,E2 -24637.116} C_VEL
LIN {X 0,Y 136.256,Z 423.517,A -85,B 0,C 180,E1 -24638.835,E2 -24638.835} C_VEL
LIN {X 0,Y 136.274,Z 423.518,A -85,B 0,C 180,E1 -24645.056,E2 -24645.056} C_VEL
LIN {X 0,Y 136.442,Z 423.497,A -85,B 0,C 180,E1 -24648.167,E2 -24648.167} C_VEL
LIN {X 0,Y 136.562,Z 423.479,A -85,B 0,C 180,E1 -24651.118,E2 -24651.118} C_VEL
LIN {X 0,Y 137.142,Z 423.402,A -85,B 0,C 180,E1 -24660,E2 -24660} C_VEL
LIN {X 0,Y 136.602,Z 423.434,A -85,B 0,C 180,E1 -24668.879,E2 -24668.879} C_VEL
LIN {X 0,Y 136.502,Z 423.477,A -85,B 0,C 180,E1 -24671.953,E2 -24671.953} C_VEL
LIN {X 0,Y 136.262,Z 423.479,A -85,B 0,C 180,E1 -24678.027,E2 -24678.027} C_VEL
LIN {X 0,Y 136.208,Z 423.481,A -85,B 0,C 180,E1 -24681.746,E2 -24681.746} C_VEL
LIN {X 0,Y 136.109,Z 423.524,A -85,B 0,C 180,E1 -24688.612,E2 -24688.612} C_VEL
LIN {X 0,Y 136.052,Z 423.508,A -85,B 0,C 180,E1 -24694.626,E2 -24694.626} C_VEL
LIN {X 0,Y 136.042,Z 423.538,A -85,B 0,C 180,E1 -24699.196,E2 -24699.196} C_VEL
LIN {X 0,Y 135.99,Z 423.515,A -85,B 0,C 180,E1 -24703.647,E2 -24703.647} C_VEL
LIN {X 0,Y 136.036,Z 423.54,A -85,B 0,C 180,E1 -24707.802,E2 -24707.802} C_VEL
LIN {X 0,Y 136.034,Z 423.521,A -85,B 0,C 180,E1 -24711.68,E2 -24711.68} C_VEL
LIN {X 0,Y 136.092,Z 423.534,A -85,B 0,C 180,E1 -24715.717,E2 -24715.717} C_VEL
LIN {X 0,Y 136.104,Z 423.532,A -85,B 0,C 180,E1 -24721.046,E2 -24721.046} C_VEL
LIN {X 0,Y 137.029,Z 426.189,A -85,B 0,C 180,E1 -24721.771,E2 -24721.771} C_VEL
LIN {X 0,Y 138.888,Z 428.715,A -85,B 0,C 180,E1 -24722.903,E2 -24722.903} C_VEL
LIN {X 0,Y 140.841,Z 432.005,A -85,B 0,C 180,E1 -24724.15,E2 -24724.15} C_VEL
LIN {X 0,Y 146.437,Z 442.379,A -85,B 0,C 180,E1 -24727.965,E2 -24727.965} C_VEL
LIN {X 0,Y 150.385,Z 451.906,A -85,B 0,C 180,E1 -24731.211,E2 -24731.211} C_VEL
LIN {X 0,Y 151.978,Z 457.537,A -85,B 0,C 180,E1 -24733.033,E2 -24733.033} C_VEL
LIN {X 0,Y 152.775,Z 464.096,A -85,B 0,C 180,E1 -24735.026,E2 -24735.026} C_VEL
LIN {X 0,Y 153.285,Z 472.924,A -85,B 0,C 180,E1 -24737.891,E2 -24737.891} C_VEL
LIN {X 0,Y 153.159,Z 474.532,A -85,B 0,C 180,E1 -24738.394,E2 -24738.394} C_VEL
LIN {X 0,Y 149.193,Z 485.07,A -85,B 0,C 180,E1 -24741.587,E2 -24741.587} C_VEL
LIN {X 0,Y 145.486,Z 494.115,A -85,B 0,C 180,E1 -24745.145,E2 -24745.145} C_VEL
LIN {X 0,Y 141.869,Z 502.211,A -85,B 0,C 180,E1 -24749.285,E2 -24749.285} C_VEL
LIN {X 0,Y 139.432,Z 507.698,A -85,B 0,C 180,E1 -24752.884,E2 -24752.884} C_VEL
LIN {X 0,Y 137.107,Z 512.995,A -85,B 0,C 180,E1 -24757.357,E2 -24757.357} C_VEL
LIN {X 0,Y 135.344,Z 517.105,A -85,B 0,C 180,E1 -24761.982,E2 -24761.982} C_VEL
LIN {X 0,Y 134.456,Z 519.239,A -85,B 0,C 180,E1 -24765.144,E2 -24765.144} C_VEL
LIN {X 0,Y 133.842,Z 521.183,A -85,B 0,C 180,E1 -24769.061,E2 -24769.061} C_VEL
LIN {X 0,Y 133.746,Z 522.805,A -85,B 0,C 180,E1 -24774.852,E2 -24774.852} C_VEL
LIN {X 0,Y 134.125,Z 523.086,A -85,B 0,C 180,E1 -24778.13,E2 -24778.13} C_VEL
LIN {X 0,Y 135.714,Z 522.37,A -85,B 0,C 180,E1 -24784.049,E2 -24784.049} C_VEL
LIN {X 0,Y 137.272,Z 521.072,A -85,B 0,C 180,E1 -24787.898,E2 -24787.898} C_VEL
LIN {X 0,Y 140,Z 518.386,A -85,B 0,C 180,E1 -24792.655,E2 -24792.655} C_VEL
LIN {X 0,Y 143.565,Z 514.464,A -85,B 0,C 180,E1 -24797.239,E2 -24797.239} C_VEL
LIN {X 0,Y 148.244,Z 508.715,A -85,B 0,C 180,E1 -24801.953,E2 -24801.953} C_VEL
LIN {X 0,Y 152.997,Z 502.238,A -85,B 0,C 180,E1 -24805.765,E2 -24805.765} C_VEL
LIN {X 0,Y 157.79,Z 494.982,A -85,B 0,C 180,E1 -24809.015,E2 -24809.015} C_VEL
LIN {X 0,Y 162.564,Z 486.928,A -85,B 0,C 180,E1 -24811.803,E2 -24811.803} C_VEL
LIN {X 0,Y 163.316,Z 485.147,A -85,B 0,C 180,E1 -24812.445,E2 -24812.445} C_VEL
LIN {X 0,Y 163.787,Z 479.083,A -85,B 0,C 180,E1 -24815.207,E2 -24815.207} C_VEL
LIN {X 0,Y 163.568,Z 473.394,A -85,B 0,C 180,E1 -24817.916,E2 -24817.916} C_VEL
LIN {X 0,Y 162.782,Z 468.547,A -85,B 0,C 180,E1 -24820.452,E2 -24820.452} C_VEL
LIN {X 0,Y 161.006,Z 462.576,A -85,B 0,C 180,E1 -24824.008,E2 -24824.008} C_VEL
LIN {X 0,Y 159.225,Z 457.84,A -85,B 0,C 180,E1 -24827.25,E2 -24827.25} C_VEL
LIN {X 0,Y 156.498,Z 451.866,A -85,B 0,C 180,E1 -24832.258,E2 -24832.258} C_VEL
LIN {X 0,Y 155.237,Z 449.394,A -85,B 0,C 180,E1 -24834.805,E2 -24834.805} C_VEL
LIN {X 0,Y 152.331,Z 444.337,A -85,B 0,C 180,E1 -24842.645,E2 -24842.645} C_VEL
LIN {X 0,Y 150.961,Z 444.233,A -85,B 0,C 180,E1 -24848.029,E2 -24848.029} C_VEL
LIN {X 0,Y 150.791,Z 445.086,A -85,B 0,C 180,E1 -24853.476,E2 -24853.476} C_VEL
LIN {X 0,Y 151.854,Z 446.84,A -85,B 0,C 180,E1 -24858.903,E2 -24858.903} C_VEL
LIN {X 0,Y 152.228,Z 447.642,A -85,B 0,C 180,E1 -24860.259,E2 -24860.259} C_VEL
LIN {X 0,Y 153.411,Z 451.635,A -85,B 0,C 180,E1 -24864.35,E2 -24864.35} C_VEL
LIN {X 0,Y 154.75,Z 453.809,A -85,B 0,C 180,E1 -24867.011,E2 -24867.011} C_VEL
LIN {X 0,Y 155.906,Z 457.61,A -85,B 0,C 180,E1 -24869.727,E2 -24869.727} C_VEL
LIN {X 0,Y 157.082,Z 460.183,A -85,B 0,C 180,E1 -24871.791,E2 -24871.791} C_VEL
LIN {X 0,Y 159.215,Z 466.718,A -85,B 0,C 180,E1 -24875.795,E2 -24875.795} C_VEL
LIN {X 0,Y 161.076,Z 473.056,A -85,B 0,C 180,E1 -24879.245,E2 -24879.245} C_VEL
LIN {X 0,Y 162.068,Z 477.898,A -85,B 0,C 180,E1 -24881.566,E2 -24881.566} C_VEL
LIN {X 0,Y 161.958,Z 481.54,A -85,B 0,C 180,E1 -24882.924,E2 -24882.924} C_VEL
LIN {X 0,Y 160.835,Z 489.421,A -85,B 0,C 180,E1 -24885.649,E2 -24885.649} C_VEL
LIN {X 0,Y 158.71,Z 498.239,A -85,B 0,C 180,E1 -24888.833,E2 -24888.833} C_VEL
LIN {X 0,Y 156.111,Z 505.681,A -85,B 0,C 180,E1 -24891.763,E2 -24891.763} C_VEL
LIN {X 0,Y 154.072,Z 510.113,A -85,B 0,C 180,E1 -24893.637,E2 -24893.637} C_VEL
LIN {X 0,Y 148.983,Z 517.737,A -85,B 0,C 180,E1 -24897.154,E2 -24897.154} C_VEL
LIN {X 0,Y 144.335,Z 524.333,A -85,B 0,C 180,E1 -24901.219,E2 -24901.219} C_VEL
LIN {X 0,Y 141.033,Z 528.907,A -85,B 0,C 180,E1 -24904.946,E2 -24904.946} C_VEL
LIN {X 0,Y 138.032,Z 532.799,A -85,B 0,C 180,E1 -24909.126,E2 -24909.126} C_VEL
LIN {X 0,Y 136.421,Z 534.836,A -85,B 0,C 180,E1 -24912.001,E2 -24912.001} C_VEL
LIN {X 0,Y 135.29,Z 536.479,A -85,B 0,C 180,E1 -24914.952,E2 -24914.952} C_VEL
LIN {X 0,Y 134.473,Z 537.712,A -85,B 0,C 180,E1 -24917.939,E2 -24917.939} C_VEL
LIN {X 0,Y 133.753,Z 538.966,A -85,B 0,C 180,E1 -24923.974,E2 -24923.974} C_VEL
LIN {X 0,Y 133.786,Z 539.022,A -85,B 0,C 180,E1 -24926.995,E2 -24926.995} C_VEL
LIN {X 0,Y 134.02,Z 538.687,A -85,B 0,C 180,E1 -24930.006,E2 -24930.006} C_VEL
LIN {X 0,Y 133.833,Z 537.566,A -85,B 0,C 180,E1 -24933.84,E2 -24933.84} C_VEL
LIN {X 0,Y 134.074,Z 534.978,A -85,B 0,C 180,E1 -24939.053,E2 -24939.053} C_VEL
LIN {X 0,Y 134.897,Z 531.623,A -85,B 0,C 180,E1 -24943.564,E2 -24943.564} C_VEL
LIN {X 0,Y 136.458,Z 527.174,A -85,B 0,C 180,E1 -24948.006,E2 -24948.006} C_VEL
LIN {X 0,Y 138.805,Z 521.515,A -85,B 0,C 180,E1 -24952.323,E2 -24952.323} C_VEL
LIN {X 0,Y 141.278,Z 515.692,A -85,B 0,C 180,E1 -24955.808,E2 -24955.808} C_VEL
LIN {X 0,Y 144.917,Z 507.169,A -85,B 0,C 180,E1 -24959.813,E2 -24959.813} C_VEL
LIN {X 0,Y 147.452,Z 500.267,A -85,B 0,C 180,E1 -24962.431,E2 -24962.431} C_VEL
LIN {X 0,Y 148.729,Z 490.844,A -85,B 0,C 180,E1 -24965.701,E2 -24965.701} C_VEL
LIN {X 0,Y 149.346,Z 481.477,A -85,B 0,C 180,E1 -24968.518,E2 -24968.518} C_VEL
LIN {X 0,Y 149.483,Z 471.16,A -85,B 0,C 180,E1 -24971.214,E2 -24971.214} C_VEL
LIN {X 0,Y 148.746,Z 459.741,A -85,B 0,C 180,E1 -24973.897,E2 -24973.897} C_VEL
LIN {X 0,Y 147.434,Z 454.065,A -85,B 0,C 180,E1 -24975.333,E2 -24975.333} C_VEL
LIN {X 0,Y 144.138,Z 445.452,A -85,B 0,C 180,E1 -24977.781,E2 -24977.781} C_VEL
LIN {X 0,Y 141.632,Z 440.263,A -85,B 0,C 180,E1 -24979.361,E2 -24979.361} C_VEL
LIN {X 0,Y 139.762,Z 436.228,A -85,B 0,C 180,E1 -24980.547,E2 -24980.547} C_VEL
LIN {X 0,Y 137.726,Z 432.595,A -85,B 0,C 180,E1 -24981.762,E2 -24981.762} C_VEL
LIN {X 0,Y 137.381,Z 431.187,A -85,B 0,C 180,E1 -24982.129,E2 -24982.129} C_VEL
LIN {X 0,Y 137.065,Z 429.259,A -85,B 0,C 180,E1 -24985.665,E2 -24985.665} C_VEL
LIN {X 0,Y 136.644,Z 426.536,A -85,B 0,C 180,E1 -24991.067,E2 -24991.067} C_VEL
LIN {X 0,Y 135.801,Z 425.582,A -85,B 0,C 180,E1 -24993.487,E2 -24993.487} C_VEL
LIN {X 0,Y 134.123,Z 424.967,A -85,B 0,C 180,E1 -24995.891,E2 -24995.891} C_VEL
LIN {X 0,Y 129.522,Z 424.416,A -85,B 0,C 180,E1 -25002.578,E2 -25002.578} C_VEL
LIN {X 0,Y 129.199,Z 424.399,A -85,B 0,C 180,E1 -25004.35,E2 -25004.35} C_VEL
LIN {X 0,Y 129.387,Z 424.375,A -85,B 0,C 180,E1 -25007.905,E2 -25007.905} C_VEL
LIN {X 0,Y 129.485,Z 424.362,A -85,B 0,C 180,E1 -25010.629,E2 -25010.629} C_VEL
LIN {X 0,Y 130.098,Z 424.28,A -85,B 0,C 180,E1 -25020,E2 -25020} C_VEL
LIN {X 0,Y 129.528,Z 424.318,A -85,B 0,C 180,E1 -25029.368,E2 -25029.368} C_VEL
LIN {X 0,Y 129.405,Z 424.365,A -85,B 0,C 180,E1 -25032.547,E2 -25032.547} C_VEL
LIN {X 0,Y 129.169,Z 424.352,A -85,B 0,C 180,E1 -25039.054,E2 -25039.054} C_VEL
LIN {X 0,Y 129.119,Z 424.368,A -85,B 0,C 180,E1 -25042.396,E2 -25042.396} C_VEL
LIN {X 0,Y 129.038,Z 424.411,A -85,B 0,C 180,E1 -25045.831,E2 -25045.831} C_VEL
LIN {X 0,Y 129.026,Z 424.399,A -85,B 0,C 180,E1 -25049.355,E2 -25049.355} C_VEL
LIN {X 0,Y 128.969,Z 424.394,A -85,B 0,C 180,E1 -25055.165,E2 -25055.165} C_VEL
LIN {X 0,Y 128.937,Z 424.412,A -85,B 0,C 180,E1 -25060.85,E2 -25060.85} C_VEL
LIN {X 0,Y 128.926,Z 424.399,A -85,B 0,C 180,E1 -25065.125,E2 -25065.125} C_VEL
LIN {X 0,Y 128.955,Z 424.417,A -85,B 0,C 180,E1 -25069.729,E2 -25069.729} C_VEL
LIN {X 0,Y 128.987,Z 424.409,A -85,B 0,C 180,E1 -25074.814,E2 -25074.814} C_VEL
LIN {X 0,Y 128.991,Z 424.415,A -85,B 0,C 180,E1 -25077.829,E2 -25077.829} C_VEL
LIN {X 0,Y 129.999,Z 427.223,A -85,B 0,C 180,E1 -25078.756,E2 -25078.756} C_VEL
LIN {X 0,Y 132.07,Z 429.808,A -85,B 0,C 180,E1 -25080.139,E2 -25080.139} C_VEL
LIN {X 0,Y 134.186,Z 433.239,A -85,B 0,C 180,E1 -25081.664,E2 -25081.664} C_VEL
LIN {X 0,Y 139.119,Z 442.46,A -85,B 0,C 180,E1 -25085.412,E2 -25085.412} C_VEL
LIN {X 0,Y 142.51,Z 449.66,A -85,B 0,C 180,E1 -25088.233,E2 -25088.233} C_VEL
LIN {X 0,Y 145.119,Z 456.94,A -85,B 0,C 180,E1 -25090.895,E2 -25090.895} C_VEL
LIN {X 0,Y 146.298,Z 462.723,A -85,B 0,C 180,E1 -25092.873,E2 -25092.873} C_VEL
LIN {X 0,Y 146.821,Z 472.498,A -85,B 0,C 180,E1 -25096.147,E2 -25096.147} C_VEL
LIN {X 0,Y 146.8,Z 475.488,A -85,B 0,C 180,E1 -25097.202,E2 -25097.202} C_VEL
LIN {X 0,Y 142.835,Z 485.544,A -85,B 0,C 180,E1 -25100.37,E2 -25100.37} C_VEL
LIN {X 0,Y 138.822,Z 494.855,A -85,B 0,C 180,E1 -25104.183,E2 -25104.183} C_VEL
LIN {X 0,Y 135.071,Z 502.87,A -85,B 0,C 180,E1 -25108.504,E2 -25108.504} C_VEL
LIN {X 0,Y 132.041,Z 509.275,A -85,B 0,C 180,E1 -25113.045,E2 -25113.045} C_VEL
LIN {X 0,Y 129.706,Z 514.341,A -85,B 0,C 180,E1 -25117.779,E2 -25117.779} C_VEL
LIN {X 0,Y 127.984,Z 518.233,A -85,B 0,C 180,E1 -25122.682,E2 -25122.682} C_VEL
LIN {X 0,Y 127.152,Z 520.229,A -85,B 0,C 180,E1 -25126.037,E2 -25126.037} C_VEL
LIN {X 0,Y 126.721,Z 521.731,A -85,B 0,C 180,E1 -25129.468,E2 -25129.468} C_VEL
LIN {X 0,Y 126.564,Z 522.784,A -85,B 0,C 180,E1 -25132.867,E2 -25132.867} C_VEL
LIN {X 0,Y 126.95,Z 523.477,A -85,B 0,C 180,E1 -25137.654,E2 -25137.654} C_VEL
LIN {X 0,Y 128.288,Z 523.189,A -85,B 0,C 180,E1 -25143.21,E2 -25143.21} C_VEL
LIN {X 0,Y 129.512,Z 522.377,A -85,B 0,C 180,E1 -25146.641,E2 -25146.641} C_VEL
LIN {X 0,Y 132.233,Z 520.105,A -85,B 0,C 180,E1 -25151.92,E2 -25151.92} C_VEL
LIN {X 0,Y 135.541,Z 516.919,A -85,B 0,C 180,E1 -25156.536,E2 -25156.536} C_VEL
LIN {X 0,Y 139.768,Z 512.296,A -85,B 0,C 180,E1 -25161.195,E2 -25161.195} C_VEL
LIN {X 0,Y 144.887,Z 506.216,A -85,B 0,C 180,E1 -25165.539,E2 -25165.539} C_VEL
LIN {X 0,Y 149.87,Z 499.46,A -85,B 0,C 180,E1 -25169.12,E2 -25169.12} C_VEL
LIN {X 0,Y 155.702,Z 490.635,A -85,B 0,C 180,E1 -25172.603,E2 -25172.603} C_VEL
LIN {X 0,Y 157.232,Z 488.068,A -85,B 0,C 180,E1 -25173.45,E2 -25173.45} C_VEL
LIN {X 0,Y 157.982,Z 484.029,A -85,B 0,C 180,E1 -25175.373,E2 -25175.373} C_VEL
LIN {X 0,Y 158.275,Z 478.909,A -85,B 0,C 180,E1 -25177.963,E2 -25177.963} C_VEL
LIN {X 0,Y 157.779,Z 473.17,A -85,B 0,C 180,E1 -25181.159,E2 -25181.159} C_VEL
LIN {X 0,Y 156.621,Z 468.131,A -85,B 0,C 180,E1 -25184.381,E2 -25184.381} C_VEL
LIN {X 0,Y 154.952,Z 462.919,A -85,B 0,C 180,E1 -25188.223,E2 -25188.223} C_VEL
LIN {X 0,Y 152.937,Z 457.792,A -85,B 0,C 180,E1 -25192.872,E2 -25192.872} C_VEL
LIN {X 0,Y 152.208,Z 456.159,A -85,B 0,C 180,E1 -25194.702,E2 -25194.702} C_VEL
LIN {X 0,Y 149.754,Z 451.024,A -85,B 0,C 180,E1 -25202.69,E2 -25202.69} C_VEL
LIN {X 0,Y 148.474,Z 450.901,A -85,B 0,C 180,E1 -25208.164,E2 -25208.164} C_VEL
LIN {X 0,Y 148.328,Z 451.837,A -85,B 0,C 180,E1 -25213.704,E2 -25213.704} C_VEL
LIN {X 0,Y 149.37,Z 453.736,A -85,B 0,C 180,E1 -25219.23,E2 -25219.23} C_VEL
LIN {X 0,Y 151.333,Z 459.744,A -85,B 0,C 180,E1 -25226.18,E2 -25226.18} C_VEL
LIN {X 0,Y 152.926,Z 464.871,A -85,B 0,C 180,E1 -25230.367,E2 -25230.367} C_VEL
LIN {X 0,Y 154.669,Z 471.174,A -85,B 0,C 180,E1 -25234.612,E2 -25234.612} C_VEL
LIN {X 0,Y 156.411,Z 478.715,A -85,B 0,C 180,E1 -25238.981,E2 -25238.981} C_VEL
LIN {X 0,Y 156.83,Z 482.335,A -85,B 0,C 180,E1 -25240.788,E2 -25240.788} C_VEL
LIN {X 0,Y 155.581,Z 490.092,A -85,B 0,C 180,E1 -25243.725,E2 -25243.725} C_VEL
LIN {X 0,Y 152.986,Z 499.398,A -85,B 0,C 180,E1 -25247.31,E2 -25247.31} C_VEL
LIN {X 0,Y 150.497,Z 506.002,A -85,B 0,C 180,E1 -25250.059,E2 -25250.059} C_VEL
LIN {X 0,Y 148.368,Z 510.327,A -85,B 0,C 180,E1 -25251.998,E2 -25251.998} C_VEL
LIN {X 0,Y 143.067,Z 517.817,A -85,B 0,C 180,E1 -25255.61,E2 -25255.61} C_VEL
LIN {X 0,Y 137.855,Z 524.676,A -85,B 0,C 180,E1 -25260.076,E2 -25260.076} C_VEL
LIN {X 0,Y 134.623,Z 528.779,A -85,B 0,C 180,E1 -25263.664,E2 -25263.664} C_VEL
LIN {X 0,Y 131.399,Z 532.593,A -85,B 0,C 180,E1 -25268.019,E2 -25268.019} C_VEL
LIN {X 0,Y 129.653,Z 534.593,A -85,B 0,C 180,E1 -25271.027,E2 -25271.027} C_VEL
LIN {X 0,Y 128.405,Z 536.195,A -85,B 0,C 180,E1 -25274.124,E2 -25274.124} C_VEL
LIN {X 0,Y 126.927,Z 538.142,A -85,B 0,C 180,E1 -25280.445,E2 -25280.445} C_VEL
LIN {X 0,Y 126.692,Z 538.548,A -85,B 0,C 180,E1 -25283.636,E2 -25283.636} C_VEL
LIN {X 0,Y 126.699,Z 538.571,A -85,B 0,C 180,E1 -25286.826,E2 -25286.826} C_VEL
LIN {X 0,Y 126.937,Z 538.181,A -85,B 0,C 180,E1 -25290.006,E2 -25290.006} C_VEL
LIN {X 0,Y 126.77,Z 537.142,A -85,B 0,C 180,E1 -25293.703,E2 -25293.703} C_VEL
LIN {X 0,Y 127.041,Z 534.364,A -85,B 0,C 180,E1 -25299.559,E2 -25299.559} C_VEL
LIN {X 0,Y 127.973,Z 530.938,A -85,B 0,C 180,E1 -25304.314,E2 -25304.314} C_VEL
LIN {X 0,Y 129.688,Z 526.414,A -85,B 0,C 180,E1 -25308.981,E2 -25308.981} C_VEL
LIN {X 0,Y 132.195,Z 520.655,A -85,B 0,C 180,E1 -25313.505,E2 -25313.505} C_VEL
LIN {X 0,Y 134.817,Z 514.747,A -85,B 0,C 180,E1 -25317.144,E2 -25317.144} C_VEL
LIN {X 0,Y 138.746,Z 506.068,A -85,B 0,C 180,E1 -25321.285,E2 -25321.285} C_VEL
LIN {X 0,Y 140.742,Z 500.9,A -85,B 0,C 180,E1 -25323.324,E2 -25323.324} C_VEL
LIN {X 0,Y 142.062,Z 492.57,A -85,B 0,C 180,E1 -25326.423,E2 -25326.423} C_VEL
LIN {X 0,Y 142.967,Z 482.336,A -85,B 0,C 180,E1 -25329.727,E2 -25329.727} C_VEL
LIN {X 0,Y 143.312,Z 471.909,A -85,B 0,C 180,E1 -25332.642,E2 -25332.642} C_VEL
LIN {X 0,Y 142.626,Z 460.453,A -85,B 0,C 180,E1 -25335.576,E2 -25335.576} C_VEL
LIN {X 0,Y 140.202,Z 452.68,A -85,B 0,C 180,E1 -25337.897,E2 -25337.897} C_VEL
LIN {X 0,Y 136.961,Z 444.934,A -85,B 0,C 180,E1 -25340.421,E2 -25340.421} C_VEL
LIN {X 0,Y 134.796,Z 440.326,A -85,B 0,C 180,E1 -25341.983,E2 -25341.983} C_VEL
LIN {X 0,Y 132.54,Z 435.858,A -85,B 0,C 180,E1 -25343.555,E2 -25343.555} C_VEL
LIN {X 0,Y 130.634,Z 432.641,A -85,B 0,C 180,E1 -25344.823,E2 -25344.823} C_VEL
LIN {X 0,Y 130.097,Z 430.632,A -85,B 0,C 180,E1 -25345.312,E2 -25345.312} C_VEL
LIN {X 0,Y 129.655,Z 427.903,A -85,B 0,C 180,E1 -25351.015,E2 -25351.015} C_VEL
LIN {X 0,Y 129.282,Z 425.05,A -85,B 0,C 180,E1 -25357.633,E2 -25357.633} C_VEL
LIN {X 0,Y 129.192,Z 424.397,A -85,B 0,C 180,E1 -25359.292,E2 -25359.292} C_VEL
LIN {X 0,Y 129.199,Z 424.399,A -85,B 0,C 180,E1 -25364.35,E2 -25364.35} C_VEL
LIN {X 0,Y 128.519,Z 424.484,A -85,B 0,C 180,E1 -25366.956,E2 -25366.956} C_VEL
LIN {X 0,Y 126.968,Z 424.676,A -85,B 0,C 180,E1 -25369.532,E2 -25369.532} C_VEL
LIN {X 0,Y 123.512,Z 425.102,A -85,B 0,C 180,E1 -25374.814,E2 -25374.814} C_VEL
LIN {X 0,Y 122.758,Z 425.194,A -85,B 0,C 180,E1 -25377.592,E2 -25377.592} C_VEL
LIN {X 0,Y 122.802,Z 425.182,A -85,B 0,C 180,E1 -25378.527,E2 -25378.527} C_VEL
LIN {X 0,Y 123.051,Z 425.158,A -85,B 0,C 180,E1 -25380,E2 -25380} C_VEL
LIN {X 0,Y 122.424,Z 425.187,A -85,B 0,C 180,E1 -25387.189,E2 -25387.189} C_VEL
LIN {X 0,Y 122.375,Z 425.239,A -85,B 0,C 180,E1 -25392.472,E2 -25392.472} C_VEL
LIN {X 0,Y 122.128,Z 425.252,A -85,B 0,C 180,E1 -25396.722,E2 -25396.722} C_VEL
LIN {X 0,Y 122.038,Z 425.253,A -85,B 0,C 180,E1 -25402.853,E2 -25402.853} C_VEL
LIN {X 0,Y 121.951,Z 425.293,A -85,B 0,C 180,E1 -25407.454,E2 -25407.454} C_VEL
LIN {X 0,Y 121.909,Z 425.262,A -85,B 0,C 180,E1 -25411.255,E2 -25411.255} C_VEL
LIN {X 0,Y 121.894,Z 425.287,A -85,B 0,C 180,E1 -25416.168,E2 -25416.168} C_VEL
LIN {X 0,Y 121.876,Z 425.282,A -85,B 0,C 180,E1 -25421.432,E2 -25421.432} C_VEL
LIN {X 0,Y 121.887,Z 425.303,A -85,B 0,C 180,E1 -25428.554,E2 -25428.554} C_VEL
LIN {X 0,Y 121.937,Z 425.425,A -85,B 0,C 180,E1 -25434.154,E2 -25434.154} C_VEL
LIN {X 0,Y 122.94,Z 428.147,A -85,B 0,C 180,E1 -25435.193,E2 -25435.193} C_VEL
LIN {X 0,Y 125.048,Z 430.594,A -85,B 0,C 180,E1 -25436.814,E2 -25436.814} C_VEL
LIN {X 0,Y 127.048,Z 434.011,A -85,B 0,C 180,E1 -25438.496,E2 -25438.496} C_VEL
LIN {X 0,Y 129.368,Z 437.807,A -85,B 0,C 180,E1 -25440.367,E2 -25440.367} C_VEL
LIN {X 0,Y 134.109,Z 446.96,A -85,B 0,C 180,E1 -25444.504,E2 -25444.504} C_VEL
LIN {X 0,Y 137.069,Z 453.675,A -85,B 0,C 180,E1 -25447.357,E2 -25447.357} C_VEL
LIN {X 0,Y 139.471,Z 460.989,A -85,B 0,C 180,E1 -25450.274,E2 -25450.274} C_VEL
LIN {X 0,Y 140.278,Z 466.152,A -85,B 0,C 180,E1 -25452.159,E2 -25452.159} C_VEL
LIN {X 0,Y 140.481,Z 475.379,A -85,B 0,C 180,E1 -25455.509,E2 -25455.509} C_VEL
LIN {X 0,Y 139.719,Z 478.467,A -85,B 0,C 180,E1 -25456.542,E2 -25456.542} C_VEL
LIN {X 0,Y 135.684,Z 487.938,A -85,B 0,C 180,E1 -25459.782,E2 -25459.782} C_VEL
LIN {X 0,Y 131.479,Z 496.97,A -85,B 0,C 180,E1 -25463.857,E2 -25463.857} C_VEL
LIN {X 0,Y 127.688,Z 504.661,A -85,B 0,C 180,E1 -25468.417,E2 -25468.417} C_VEL
LIN {X 0,Y 124.64,Z 510.813,A -85,B 0,C 180,E1 -25473.226,E2 -25473.226} C_VEL
LIN {X 0,Y 122.346,Z 515.63,A -85,B 0,C 180,E1 -25478.25,E2 -25478.25} C_VEL
LIN {X 0,Y 120.616,Z 519.304,A -85,B 0,C 180,E1 -25483.471,E2 -25483.471} C_VEL
LIN {X 0,Y 119.601,Z 522.271,A -85,B 0,C 180,E1 -25489.917,E2 -25489.917} C_VEL
LIN {X 0,Y 119.51,Z 523.443,A -85,B 0,C 180,E1 -25494.301,E2 -25494.301} C_VEL
LIN {X 0,Y 120.008,Z 523.936,A -85,B 0,C 180,E1 -25498.545,E2 -25498.545} C_VEL
LIN {X 0,Y 120.66,Z 523.919,A -85,B 0,C 180,E1 -25501.607,E2 -25501.607} C_VEL
LIN {X 0,Y 122.241,Z 523.184,A -85,B 0,C 180,E1 -25506.4,E2 -25506.4} C_VEL
LIN {X 0,Y 125.183,Z 521.077,A -85,B 0,C 180,E1 -25512.344,E2 -25512.344} C_VEL
LIN {X 0,Y 128.823,Z 517.931,A -85,B 0,C 180,E1 -25517.424,E2 -25517.424} C_VEL
LIN {X 0,Y 133.243,Z 513.491,A -85,B 0,C 180,E1 -25522.285,E2 -25522.285} C_VEL
LIN {X 0,Y 138.654,Z 507.552,A -85,B 0,C 180,E1 -25526.832,E2 -25526.832} C_VEL
LIN {X 0,Y 144.508,Z 500.22,A -85,B 0,C 180,E1 -25530.9,E2 -25530.9} C_VEL
LIN {X 0,Y 150.037,Z 492.36,A -85,B 0,C 180,E1 -25534.128,E2 -25534.128} C_VEL
LIN {X 0,Y 151.04,Z 490.876,A -85,B 0,C 180,E1 -25534.637,E2 -25534.637} C_VEL
LIN {X 0,Y 151.891,Z 489.07,A -85,B 0,C 180,E1 -25535.391,E2 -25535.391} C_VEL
LIN {X 0,Y 152.723,Z 483.508,A -85,B 0,C 180,E1 -25538.399,E2 -25538.399} C_VEL
LIN {X 0,Y 152.753,Z 478.711,A -85,B 0,C 180,E1 -25541.212,E2 -25541.212} C_VEL
LIN {X 0,Y 151.832,Z 472.84,A -85,B 0,C 180,E1 -25545.251,E2 -25545.251} C_VEL
LIN {X 0,Y 150.542,Z 467.927,A -85,B 0,C 180,E1 -25549.238,E2 -25549.238} C_VEL
LIN {X 0,Y 149.219,Z 463.793,A -85,B 0,C 180,E1 -25553.238,E2 -25553.238} C_VEL
LIN {X 0,Y 147.647,Z 460.184,A -85,B 0,C 180,E1 -25558.171,E2 -25558.171} C_VEL
LIN {X 0,Y 146.819,Z 457.557,A -85,B 0,C 180,E1 -25562.744,E2 -25562.744} C_VEL
LIN {X 0,Y 145.637,Z 457.426,A -85,B 0,C 180,E1 -25568.324,E2 -25568.324} C_VEL
LIN {X 0,Y 145.518,Z 458.439,A -85,B 0,C 180,E1 -25573.974,E2 -25573.974} C_VEL
LIN {X 0,Y 145.892,Z 459.291,A -85,B 0,C 180,E1 -25576.801,E2 -25576.801} C_VEL
LIN {X 0,Y 146.376,Z 460.822,A -85,B 0,C 180,E1 -25579.639,E2 -25579.639} C_VEL
LIN {X 0,Y 147.679,Z 465.516,A -85,B 0,C 180,E1 -25585.36,E2 -25585.36} C_VEL
LIN {X 0,Y 149.042,Z 471.245,A -85,B 0,C 180,E1 -25590.251,E2 -25590.251} C_VEL
LIN {X 0,Y 150.206,Z 476.743,A -85,B 0,C 180,E1 -25594.158,E2 -25594.158} C_VEL
LIN {X 0,Y 151.248,Z 482.615,A -85,B 0,C 180,E1 -25597.83,E2 -25597.83} C_VEL
LIN {X 0,Y 151.488,Z 485.854,A -85,B 0,C 180,E1 -25599.635,E2 -25599.635} C_VEL
LIN {X 0,Y 149.969,Z 492.801,A -85,B 0,C 180,E1 -25602.44,E2 -25602.44} C_VEL
LIN {X 0,Y 147.403,Z 500.575,A -85,B 0,C 180,E1 -25605.659,E2 -25605.659} C_VEL
LIN {X 0,Y 144.274,Z 507.747,A -85,B 0,C 180,E1 -25608.889,E2 -25608.889} C_VEL
LIN {X 0,Y 141.924,Z 511.885,A -85,B 0,C 180,E1 -25610.857,E2 -25610.857} C_VEL
LIN {X 0,Y 136.377,Z 519.027,A -85,B 0,C 180,E1 -25614.574,E2 -25614.574} C_VEL
LIN {X 0,Y 131.424,Z 525.015,A -85,B 0,C 180,E1 -25618.828,E2 -25618.828} C_VEL
LIN {X 0,Y 126.997,Z 530.029,A -85,B 0,C 180,E1 -25623.73,E2 -25623.73} C_VEL
LIN {X 0,Y 124.824,Z 532.4,A -85,B 0,C 180,E1 -25626.796,E2 -25626.796} C_VEL
LIN {X 0,Y 122.935,Z 534.356,A -85,B 0,C 180,E1 -25629.947,E2 -25629.947} C_VEL
LIN {X 0,Y 120.54,Z 537.011,A -85,B 0,C 180,E1 -25636.52,E2 -25636.52} C_VEL
LIN {X 0,Y 119.631,Z 538.13,A -85,B 0,C 180,E1 -25643.259,E2 -25643.259} C_VEL
LIN {X 0,Y 119.634,Z 538.066,A -85,B 0,C 180,E1 -25647.061,E2 -25647.061} C_VEL
LIN {X 0,Y 119.855,Z 537.66,A -85,B 0,C 180,E1 -25650.006,E2 -25650.006} C_VEL
LIN {X 0,Y 119.706,Z 536.71,A -85,B 0,C 180,E1 -25653.542,E2 -25653.542} C_VEL
LIN {X 0,Y 119.72,Z 535.458,A -85,B 0,C 180,E1 -25656.749,E2 -25656.749} C_VEL
LIN {X 0,Y 120.303,Z 532.651,A -85,B 0,C 180,E1 -25661.805,E2 -25661.805} C_VEL
LIN {X 0,Y 121.61,Z 528.789,A -85,B 0,C 180,E1 -25666.802,E2 -25666.802} C_VEL
LIN {X 0,Y 123.837,Z 523.791,A -85,B 0,C 180,E1 -25671.653,E2 -25671.653} C_VEL
LIN {X 0,Y 126.839,Z 517.492,A -85,B 0,C 180,E1 -25676.319,E2 -25676.319} C_VEL
LIN {X 0,Y 129.531,Z 511.583,A -85,B 0,C 180,E1 -25679.759,E2 -25679.759} C_VEL
LIN {X 0,Y 133.422,Z 503.275,A -85,B 0,C 180,E1 -25683.585,E2 -25683.585} C_VEL
LIN {X 0,Y 134.467,Z 499.607,A -85,B 0,C 180,E1 -25685.1,E2 -25685.1} C_VEL
LIN {X 0,Y 135.972,Z 490.157,A -85,B 0,C 180,E1 -25688.711,E2 -25688.711} C_VEL
LIN {X 0,Y 136.934,Z 479.543,A -85,B 0,C 180,E1 -25692.179,E2 -25692.179} C_VEL
LIN {X 0,Y 137.121,Z 469.091,A -85,B 0,C 180,E1 -25695.191,E2 -25695.191} C_VEL
LIN {X 0,Y 136.71,Z 462.774,A -85,B 0,C 180,E1 -25696.926,E2 -25696.926} C_VEL
LIN {X 0,Y 134.253,Z 454.645,A -85,B 0,C 180,E1 -25699.65,E2 -25699.65} C_VEL
LIN {X 0,Y 130.154,Z 444.962,A -85,B 0,C 180,E1 -25703.199,E2 -25703.199} C_VEL
LIN {X 0,Y 128.02,Z 440.523,A -85,B 0,C 180,E1 -25704.92,E2 -25704.92} C_VEL
LIN {X 0,Y 126.191,Z 436.915,A -85,B 0,C 180,E1 -25706.395,E2 -25706.395} C_VEL
LIN {X 0,Y 125.429,Z 435.361,A -85,B 0,C 180,E1 -25707.005,E2 -25707.005} C_VEL
LIN {X 0,Y 123.392,Z 432.181,A -85,B 0,C 180,E1 -25708.566,E2 -25708.566} C_VEL
LIN {X 0,Y 122.753,Z 430.041,A -85,B 0,C 180,E1 -25709.192,E2 -25709.192} C_VEL
LIN {X 0,Y 122.541,Z 428.533,A -85,B 0,C 180,E1 -25712.689,E2 -25712.689} C_VEL
LIN {X 0,Y 122.35,Z 426.85,A -85,B 0,C 180,E1 -25716.803,E2 -25716.803} C_VEL
LIN {X 0,Y 122.101,Z 425.283,A -85,B 0,C 180,E1 -25721.544,E2 -25721.544} C_VEL
LIN {X 0,Y 122.325,Z 425.255,A -85,B 0,C 180,E1 -25727.634,E2 -25727.634} C_VEL
LIN {X 0,Y 122.434,Z 425.238,A -85,B 0,C 180,E1 -25733.407,E2 -25733.407} C_VEL
LIN {X 0,Y 122.802,Z 425.182,A -85,B 0,C 180,E1 -25738.527,E2 -25738.527} C_VEL
LIN {X 0,Y 122.678,Z 425.204,A -85,B 0,C 180,E1 -25740.349,E2 -25740.349} C_VEL
LIN {X 0,Y 121.43,Z 425.358,A -85,B 0,C 180,E1 -25743.054,E2 -25743.054} C_VEL
LIN {X 0,Y 118.051,Z 425.781,A -85,B 0,C 180,E1 -25747.576,E2 -25747.576} C_VEL
LIN {X 0,Y 115.402,Z 426.108,A -85,B 0,C 180,E1 -25752.408,E2 -25752.408} C_VEL
LIN {X 0,Y 115.22,Z 426.131,A -85,B 0,C 180,E1 -25753.416,E2 -25753.416} C_VEL
LIN {X 0,Y 115.028,Z 426.12,A -85,B 0,C 180,E1 -25757.787,E2 -25757.787} C_VEL
LIN {X 0,Y 114.957,Z 426.141,A -85,B 0,C 180,E1 -25763.49,E2 -25763.49} C_VEL
LIN {X 0,Y 114.866,Z 426.14,A -85,B 0,C 180,E1 -25771.054,E2 -25771.054} C_VEL
LIN {X 0,Y 114.789,Z 426.185,A -85,B 0,C 180,E1 -25777.752,E2 -25777.752} C_VEL
LIN {X 0,Y 114.79,Z 426.155,A -85,B 0,C 180,E1 -25782.71,E2 -25782.71} C_VEL
LIN {X 0,Y 114.855,Z 426.334,A -85,B 0,C 180,E1 -25789.663,E2 -25789.663} C_VEL
LIN {X 0,Y 115.718,Z 428.819,A -85,B 0,C 180,E1 -25790.762,E2 -25790.762} C_VEL
LIN {X 0,Y 117.718,Z 431.044,A -85,B 0,C 180,E1 -25792.581,E2 -25792.581} C_VEL
LIN {X 0,Y 118.345,Z 431.92,A -85,B 0,C 180,E1 -25793.159,E2 -25793.159} C_VEL
LIN {X 0,Y 120.178,Z 435.044,A -85,B 0,C 180,E1 -25794.957,E2 -25794.957} C_VEL
LIN {X 0,Y 121.404,Z 436.843,A -85,B 0,C 180,E1 -25796.079,E2 -25796.079} C_VEL
LIN {X 0,Y 125.165,Z 443.359,A -85,B 0,C 180,E1 -25799.639,E2 -25799.639} C_VEL
LIN {X 0,Y 129.295,Z 452.004,A -85,B 0,C 180,E1 -25803.862,E2 -25803.862} C_VEL
LIN {X 0,Y 132.216,Z 459.557,A -85,B 0,C 180,E1 -25807.316,E2 -25807.316} C_VEL
LIN {X 0,Y 133.973,Z 466.549,A -85,B 0,C 180,E1 -25810.263,E2 -25810.263} C_VEL
LIN {X 0,Y 134.112,Z 476.027,A -85,B 0,C 180,E1 -25813.924,E2 -25813.924} C_VEL
LIN {X 0,Y 133.918,Z 478.163,A -85,B 0,C 180,E1 -25814.782,E2 -25814.782} C_VEL
LIN {X 0,Y 129.434,Z 488.329,A -85,B 0,C 180,E1 -25818.348,E2 -25818.348} C_VEL
LIN {X 0,Y 124.876,Z 497.624,A -85,B 0,C 180,E1 -25822.719,E2 -25822.719} C_VEL
LIN {X 0,Y 120.963,Z 505.128,A -85,B 0,C 180,E1 -25827.386,E2 -25827.386} C_VEL
LIN {X 0,Y 118.165,Z 510.448,A -85,B 0,C 180,E1 -25831.698,E2 -25831.698} C_VEL
LIN {X 0,Y 115.617,Z 515.455,A -85,B 0,C 180,E1 -25836.976,E2 -25836.976} C_VEL
LIN {X 0,Y 113.73,Z 519.299,A -85,B 0,C 180,E1 -25842.484,E2 -25842.484} C_VEL
LIN {X 0,Y 112.663,Z 522.04,A -85,B 0,C 180,E1 -25848.166,E2 -25848.166} C_VEL
LIN {X 0,Y 112.392,Z 523.272,A -85,B 0,C 180,E1 -25852.028,E2 -25852.028} C_VEL
LIN {X 0,Y 112.53,Z 524.057,A -85,B 0,C 180,E1 -25855.916,E2 -25855.916} C_VEL
LIN {X 0,Y 113.125,Z 524.41,A -85,B 0,C 180,E1 -25859.794,E2 -25859.794} C_VEL
LIN {X 0,Y 114.109,Z 524.26,A -85,B 0,C 180,E1 -25863.654,E2 -25863.654} C_VEL
LIN {X 0,Y 115.579,Z 523.604,A -85,B 0,C 180,E1 -25867.769,E2 -25867.769} C_VEL
LIN {X 0,Y 117.229,Z 522.604,A -85,B 0,C 180,E1 -25871.249,E2 -25871.249} C_VEL
LIN {X 0,Y 119.663,Z 520.847,A -85,B 0,C 180,E1 -25875.188,E2 -25875.188} C_VEL
LIN {X 0,Y 123.579,Z 517.632,A -85,B 0,C 180,E1 -25880.141,E2 -25880.141} C_VEL
LIN {X 0,Y 128.526,Z 512.963,A -85,B 0,C 180,E1 -25885.095,E2 -25885.095} C_VEL
LIN {X 0,Y 134.395,Z 506.815,A -85,B 0,C 180,E1 -25889.624,E2 -25889.624} C_VEL
LIN {X 0,Y 140.965,Z 498.88,A -85,B 0,C 180,E1 -25893.806,E2 -25893.806} C_VEL
LIN {X 0,Y 145.721,Z 492.385,A -85,B 0,C 180,E1 -25896.383,E2 -25896.383} C_VEL
LIN {X 0,Y 146.529,Z 490.345,A -85,B 0,C 180,E1 -25897.437,E2 -25897.437} C_VEL
LIN {X 0,Y 147.341,Z 485.236,A -85,B 0,C 180,E1 -25900.495,E2 -25900.495} C_VEL
LIN {X 0,Y 147.342,Z 481.028,A -85,B 0,C 180,E1 -25903.37,E2 -25903.37} C_VEL
LIN {X 0,Y 146.691,Z 476.242,A -85,B 0,C 180,E1 -25907.161,E2 -25907.161} C_VEL
LIN {X 0,Y 145.683,Z 471.414,A -85,B 0,C 180,E1 -25911.679,E2 -25911.679} C_VEL
LIN {X 0,Y 145.038,Z 468.939,A -85,B 0,C 180,E1 -25914.439,E2 -25914.439} C_VEL
LIN {X 0,Y 143.784,Z 465.387,A -85,B 0,C 180,E1 -25920,E2 -25920} C_VEL
LIN {X 0,Y 143.493,Z 463.902,A -85,B 0,C 180,E1 -25922.808,E2 -25922.808} C_VEL
LIN {X 0,Y 142.375,Z 463.871,A -85,B 0,C 180,E1 -25929.2,E2 -25929.2} C_VEL
LIN {X 0,Y 142.35,Z 464.89,A -85,B 0,C 180,E1 -25934.292,E2 -25934.292} C_VEL
LIN {X 0,Y 142.652,Z 465.902,A -85,B 0,C 180,E1 -25937.194,E2 -25937.194} C_VEL
LIN {X 0,Y 142.984,Z 468.416,A -85,B 0,C 180,E1 -25940.968,E2 -25940.968} C_VEL
LIN {X 0,Y 143.852,Z 471.655,A -85,B 0,C 180,E1 -25945.06,E2 -25945.06} C_VEL
LIN {X 0,Y 144.608,Z 476.016,A -85,B 0,C 180,E1 -25949.079,E2 -25949.079} C_VEL
LIN {X 0,Y 145.455,Z 481.562,A -85,B 0,C 180,E1 -25953.35,E2 -25953.35} C_VEL
LIN {X 0,Y 146.079,Z 486.911,A -85,B 0,C 180,E1 -25956.97,E2 -25956.97} C_VEL
LIN {X 0,Y 145.965,Z 490.024,A -85,B 0,C 180,E1 -25958.751,E2 -25958.751} C_VEL
LIN {X 0,Y 143.768,Z 497.08,A -85,B 0,C 180,E1 -25961.815,E2 -25961.815} C_VEL
LIN {X 0,Y 140.35,Z 505.193,A -85,B 0,C 180,E1 -25965.498,E2 -25965.498} C_VEL
LIN {X 0,Y 137.322,Z 510.803,A -85,B 0,C 180,E1 -25968.301,E2 -25968.301} C_VEL
LIN {X 0,Y 133.516,Z 515.797,A -85,B 0,C 180,E1 -25970.836,E2 -25970.836} C_VEL
LIN {X 0,Y 127.985,Z 522.069,A -85,B 0,C 180,E1 -25974.798,E2 -25974.798} C_VEL
LIN {X 0,Y 123.407,Z 527.132,A -85,B 0,C 180,E1 -25979.174,E2 -25979.174} C_VEL
LIN {X 0,Y 119.419,Z 531.118,A -85,B 0,C 180,E1 -25983.815,E2 -25983.815} C_VEL
LIN {X 0,Y 116.268,Z 534.119,A -85,B 0,C 180,E1 -25988.743,E2 -25988.743} C_VEL
LIN {X 0,Y 113.619,Z 536.668,A -85,B 0,C 180,E1 -25995.682,E2 -25995.682} C_VEL
LIN {X 0,Y 112.569,Z 537.711,A -85,B 0,C 180,E1 -26002.834,E2 -26002.834} C_VEL
LIN {X 0,Y 112.578,Z 537.539,A -85,B 0,C 180,E1 -26007.259,E2 -26007.259} C_VEL
LIN {X 0,Y 112.775,Z 537.14,A -85,B 0,C 180,E1 -26010.007,E2 -26010.007} C_VEL
LIN {X 0,Y 112.629,Z 536.21,A -85,B 0,C 180,E1 -26013.584,E2 -26013.584} C_VEL
LIN {X 0,Y 112.663,Z 534.865,A -85,B 0,C 180,E1 -26017.174,E2 -26017.174} C_VEL
LIN {X 0,Y 113.342,Z 531.984,A -85,B 0,C 180,E1 -26022.541,E2 -26022.541} C_VEL
LIN {X 0,Y 114.776,Z 528.039,A -85,B 0,C 180,E1 -26027.835,E2 -26027.835} C_VEL
LIN {X 0,Y 117.7,Z 521.965,A -85,B 0,C 180,E1 -26033.776,E2 -26033.776} C_VEL
LIN {X 0,Y 121.239,Z 514.795,A -85,B 0,C 180,E1 -26038.946,E2 -26038.946} C_VEL
LIN {X 0,Y 125.114,Z 507.14,A -85,B 0,C 180,E1 -26043.119,E2 -26043.119} C_VEL
LIN {X 0,Y 127.444,Z 502.059,A -85,B 0,C 180,E1 -26045.389,E2 -26045.389} C_VEL
LIN {X 0,Y 129.067,Z 494.11,A -85,B 0,C 180,E1 -26048.777,E2 -26048.777} C_VEL
LIN {X 0,Y 130.372,Z 484.331,A -85,B 0,C 180,E1 -26052.369,E2 -26052.369} C_VEL
LIN {X 0,Y 131.09,Z 473.566,A -85,B 0,C 180,E1 -26055.816,E2 -26055.816} C_VEL
LIN {X 0,Y 131.04,Z 466.565,A -85,B 0,C 180,E1 -26057.903,E2 -26057.903} C_VEL
LIN {X 0,Y 129.05,Z 458.781,A -85,B 0,C 180,E1 -26060.721,E2 -26060.721} C_VEL
LIN {X 0,Y 125.826,Z 450.212,A -85,B 0,C 180,E1 -26064.092,E2 -26064.092} C_VEL
LIN {X 0,Y 122.979,Z 444.201,A -85,B 0,C 180,E1 -26066.752,E2 -26066.752} C_VEL
LIN {X 0,Y 121.125,Z 440.224,A -85,B 0,C 180,E1 -26068.519,E2 -26068.519} C_VEL
LIN {X 0,Y 119.155,Z 436.415,A -85,B 0,C 180,E1 -26070.351,E2 -26070.351} C_VEL
LIN {X 0,Y 118.41,Z 435.077,A -85,B 0,C 180,E1 -26071.02,E2 -26071.02} C_VEL
LIN {X 0,Y 116.393,Z 432.04,A -85,B 0,C 180,E1 -26072.829,E2 -26072.829} C_VEL
LIN {X 0,Y 115.484,Z 429.405,A -85,B 0,C 180,E1 -26073.94,E2 -26073.94} C_VEL
LIN {X 0,Y 115.293,Z 427.633,A -85,B 0,C 180,E1 -26078.546,E2 -26078.546} C_VEL
LIN {X 0,Y 115.078,Z 426.159,A -85,B 0,C 180,E1 -26083.136,E2 -26083.136} C_VEL
LIN {X 0,Y 115.335,Z 426.124,A -85,B 0,C 180,E1 -26089.466,E2 -26089.466} C_VEL
LIN {X 0,Y 115.531,Z 426.094,A -85,B 0,C 180,E1 -26096.512,E2 -26096.512} C_VEL
LIN {X 0,Y 116.003,Z 426.035,A -85,B 0,C 180,E1 -26100,E2 -26100} C_VEL
LIN {X 0,Y 115.391,Z 426.061,A -85,B 0,C 180,E1 -26107.082,E2 -26107.082} C_VEL
LIN {X 0,Y 115.296,Z 426.122,A -85,B 0,C 180,E1 -26112.736,E2 -26112.736} C_VEL
LIN {X 0,Y 115.22,Z 426.131,A -85,B 0,C 180,E1 -26113.416,E2 -26113.416} C_VEL
LIN {X 0,Y 114.322,Z 426.245,A -85,B 0,C 180,E1 -26116.329,E2 -26116.329} C_VEL
LIN {X 0,Y 112.606,Z 426.464,A -85,B 0,C 180,E1 -26119.206,E2 -26119.206} C_VEL
LIN {X 0,Y 107.998,Z 427.032,A -85,B 0,C 180,E1 -26127.223,E2 -26127.223} C_VEL
LIN {X 0,Y 107.708,Z 427.038,A -85,B 0,C 180,E1 -26129.355,E2 -26129.355} C_VEL
LIN {X 0,Y 107.789,Z 427.015,A -85,B 0,C 180,E1 -26132.035,E2 -26132.035} C_VEL
LIN {X 0,Y 107.698,Z 427.07,A -85,B 0,C 180,E1 -26138.447,E2 -26138.447} C_VEL
LIN {X 0,Y 107.694,Z 427.036,A -85,B 0,C 180,E1 -26143.795,E2 -26143.795} C_VEL
LIN {X 0,Y 108.493,Z 429.571,A -85,B 0,C 180,E1 -26145.183,E2 -26145.183} C_VEL
LIN {X 0,Y 110.453,Z 431.792,A -85,B 0,C 180,E1 -26147.431,E2 -26147.431} C_VEL
LIN {X 0,Y 111.447,Z 432.702,A -85,B 0,C 180,E1 -26148.448,E2 -26148.448} C_VEL
LIN {X 0,Y 113.132,Z 435.866,A -85,B 0,C 180,E1 -26150.559,E2 -26150.559} C_VEL
LIN {X 0,Y 114.667,Z 437.785,A -85,B 0,C 180,E1 -26152.138,E2 -26152.138} C_VEL
LIN {X 0,Y 118.957,Z 445.093,A -85,B 0,C 180,E1 -26156.825,E2 -26156.825} C_VEL
LIN {X 0,Y 122.944,Z 453.507,A -85,B 0,C 180,E1 -26161.455,E2 -26161.455} C_VEL
LIN {X 0,Y 125.819,Z 460.854,A -85,B 0,C 180,E1 -26165.212,E2 -26165.212} C_VEL
LIN {X 0,Y 127.767,Z 468.085,A -85,B 0,C 180,E1 -26168.635,E2 -26168.635} C_VEL
LIN {X 0,Y 127.985,Z 473.161,A -85,B 0,C 180,E1 -26170.757,E2 -26170.757} C_VEL
LIN {X 0,Y 127.627,Z 479.351,A -85,B 0,C 180,E1 -26173.36,E2 -26173.36} C_VEL
LIN {X 0,Y 123.243,Z 488.772,A -85,B 0,C 180,E1 -26176.808,E2 -26176.808} C_VEL
LIN {X 0,Y 119.098,Z 496.835,A -85,B 0,C 180,E1 -26180.654,E2 -26180.654} C_VEL
LIN {X 0,Y 114.789,Z 504.694,A -85,B 0,C 180,E1 -26185.604,E2 -26185.604} C_VEL
LIN {X 0,Y 111.789,Z 510.051,A -85,B 0,C 180,E1 -26189.993,E2 -26189.993} C_VEL
LIN {X 0,Y 108.977,Z 515.225,A -85,B 0,C 180,E1 -26195.544,E2 -26195.544} C_VEL
LIN {X 0,Y 106.903,Z 519.223,A -85,B 0,C 180,E1 -26201.367,E2 -26201.367} C_VEL
LIN {X 0,Y 105.935,Z 521.304,A -85,B 0,C 180,E1 -26205.381,E2 -26205.381} C_VEL
LIN {X 0,Y 105.331,Z 523.312,A -85,B 0,C 180,E1 -26210.913,E2 -26210.913} C_VEL
LIN {X 0,Y 105.667,Z 524.661,A -85,B 0,C 180,E1 -26217.739,E2 -26217.739} C_VEL
LIN {X 0,Y 106.452,Z 524.843,A -85,B 0,C 180,E1 -26221.872,E2 -26221.872} C_VEL
LIN {X 0,Y 109.001,Z 524.022,A -85,B 0,C 180,E1 -26229.312,E2 -26229.312} C_VEL
LIN {X 0,Y 111.414,Z 522.632,A -85,B 0,C 180,E1 -26233.927,E2 -26233.927} C_VEL
LIN {X 0,Y 115.47,Z 519.856,A -85,B 0,C 180,E1 -26239.523,E2 -26239.523} C_VEL
LIN {X 0,Y 120.364,Z 515.844,A -85,B 0,C 180,E1 -26244.818,E2 -26244.818} C_VEL
LIN {X 0,Y 126.863,Z 509.819,A -85,B 0,C 180,E1 -26250.094,E2 -26250.094} C_VEL
LIN {X 0,Y 132.848,Z 503.415,A -85,B 0,C 180,E1 -26254.056,E2 -26254.056} C_VEL
LIN {X 0,Y 138.88,Z 496.07,A -85,B 0,C 180,E1 -26257.431,E2 -26257.431} C_VEL
LIN {X 0,Y 140.154,Z 494.447,A -85,B 0,C 180,E1 -26258.058,E2 -26258.058} C_VEL
LIN {X 0,Y 140.9,Z 492.865,A -85,B 0,C 180,E1 -26258.885,E2 -26258.885} C_VEL
LIN {X 0,Y 141.849,Z 488.614,A -85,B 0,C 180,E1 -26261.708,E2 -26261.708} C_VEL
LIN {X 0,Y 142.061,Z 485.268,A -85,B 0,C 180,E1 -26264.211,E2 -26264.211} C_VEL
LIN {X 0,Y 141.712,Z 480.354,A -85,B 0,C 180,E1 -26268.558,E2 -26268.558} C_VEL
LIN {X 0,Y 141.145,Z 476.216,A -85,B 0,C 180,E1 -26272.849,E2 -26272.849} C_VEL
LIN {X 0,Y 140.94,Z 475.025,A -85,B 0,C 180,E1 -26274.277,E2 -26274.277} C_VEL
LIN {X 0,Y 140.01,Z 471.515,A -85,B 0,C 180,E1 -26280,E2 -26280} C_VEL
LIN {X 0,Y 139.82,Z 470.062,A -85,B 0,C 180,E1 -26282.881,E2 -26282.881} C_VEL
LIN {X 0,Y 138.871,Z 469.988,A -85,B 0,C 180,E1 -26288.733,E2 -26288.733} C_VEL
LIN {X 0,Y 138.776,Z 471.192,A -85,B 0,C 180,E1 -26294.668,E2 -26294.668} C_VEL
LIN {X 0,Y 138.972,Z 472.422,A -85,B 0,C 180,E1 -26297.664,E2 -26297.664} C_VEL
LIN {X 0,Y 139.547,Z 476.677,A -85,B 0,C 180,E1 -26303.76,E2 -26303.76} C_VEL
LIN {X 0,Y 140.144,Z 481.841,A -85,B 0,C 180,E1 -26308.922,E2 -26308.922} C_VEL
LIN {X 0,Y 140.587,Z 487.314,A -85,B 0,C 180,E1 -26313.36,E2 -26313.36} C_VEL
LIN {X 0,Y 140.719,Z 492.38,A -85,B 0,C 180,E1 -26316.967,E2 -26316.967} C_VEL
LIN {X 0,Y 139.395,Z 496.443,A -85,B 0,C 180,E1 -26318.924,E2 -26318.924} C_VEL
LIN {X 0,Y 135.911,Z 504.253,A -85,B 0,C 180,E1 -26322.653,E2 -26322.653} C_VEL
LIN {X 0,Y 132.005,Z 511.082,A -85,B 0,C 180,E1 -26326.211,E2 -26326.211} C_VEL
LIN {X 0,Y 129.129,Z 514.807,A -85,B 0,C 180,E1 -26328.195,E2 -26328.195} C_VEL
LIN {X 0,Y 124.111,Z 520.2,A -85,B 0,C 180,E1 -26331.481,E2 -26331.481} C_VEL
LIN {X 0,Y 118.729,Z 525.681,A -85,B 0,C 180,E1 -26335.967,E2 -26335.967} C_VEL
LIN {X 0,Y 114.405,Z 529.764,A -85,B 0,C 180,E1 -26340.573,E2 -26340.573} C_VEL
LIN {X 0,Y 111.856,Z 532.04,A -85,B 0,C 180,E1 -26343.916,E2 -26343.916} C_VEL
LIN {X 0,Y 107.926,Z 535.28,A -85,B 0,C 180,E1 -26351.006,E2 -26351.006} C_VEL
LIN {X 0,Y 105.893,Z 536.998,A -85,B 0,C 180,E1 -26358.523,E2 -26358.523} C_VEL
LIN {X 0,Y 105.503,Z 537.271,A -85,B 0,C 180,E1 -26362.351,E2 -26362.351} C_VEL
LIN {X 0,Y 105.512,Z 536.992,A -85,B 0,C 180,E1 -26367.613,E2 -26367.613} C_VEL
LIN {X 0,Y 105.698,Z 536.611,A -85,B 0,C 180,E1 -26370.007,E2 -26370.007} C_VEL
LIN {X 0,Y 105.539,Z 535.642,A -85,B 0,C 180,E1 -26373.825,E2 -26373.825} C_VEL
LIN {X 0,Y 105.607,Z 534.242,A -85,B 0,C 180,E1 -26377.656,E2 -26377.656} C_VEL
LIN {X 0,Y 106.379,Z 531.288,A -85,B 0,C 180,E1 -26383.377,E2 -26383.377} C_VEL
LIN {X 0,Y 107.99,Z 527.258,A -85,B 0,C 180,E1 -26388.997,E2 -26388.997} C_VEL
LIN {X 0,Y 111.189,Z 521.051,A -85,B 0,C 180,E1 -26395.262,E2 -26395.262} C_VEL
LIN {X 0,Y 114.826,Z 514.112,A -85,B 0,C 180,E1 -26400.451,E2 -26400.451} C_VEL
LIN {X 0,Y 119.28,Z 505.828,A -85,B 0,C 180,E1 -26405.07,E2 -26405.07} C_VEL
LIN {X 0,Y 120.84,Z 502.537,A -85,B 0,C 180,E1 -26406.601,E2 -26406.601} C_VEL
LIN {X 0,Y 122.58,Z 494.936,A -85,B 0,C 180,E1 -26410.055,E2 -26410.055} C_VEL
LIN {X 0,Y 124.16,Z 485.187,A -85,B 0,C 180,E1 -26413.907,E2 -26413.907} C_VEL
LIN {X 0,Y 125.149,Z 474.341,A -85,B 0,C 180,E1 -26417.632,E2 -26417.632} C_VEL
LIN {X 0,Y 125.254,Z 469.949,A -85,B 0,C 180,E1 -26419.055,E2 -26419.055} C_VEL
LIN {X 0,Y 124.28,Z 464.819,A -85,B 0,C 180,E1 -26421.015,E2 -26421.015} C_VEL
LIN {X 0,Y 120.875,Z 454.418,A -85,B 0,C 180,E1 -26425.466,E2 -26425.466} C_VEL
LIN {X 0,Y 116.907,Z 445.225,A -85,B 0,C 180,E1 -26429.894,E2 -26429.894} C_VEL
LIN {X 0,Y 114.552,Z 440.396,A -85,B 0,C 180,E1 -26432.48,E2 -26432.48} C_VEL
LIN {X 0,Y 112.481,Z 436.588,A -85,B 0,C 180,E1 -26434.779,E2 -26434.779} C_VEL
LIN {X 0,Y 111.772,Z 434.947,A -85,B 0,C 180,E1 -26435.637,E2 -26435.637} C_VEL
LIN {X 0,Y 109.297,Z 431.569,A -85,B 0,C 180,E1 -26438.3,E2 -26438.3} C_VEL
LIN {X 0,Y 108.234,Z 428.655,A -85,B 0,C 180,E1 -26439.82,E2 -26439.82} C_VEL
LIN {X 0,Y 108.077,Z 427.031,A -85,B 0,C 180,E1 -26445.608,E2 -26445.608} C_VEL
LIN {X 0,Y 108.263,Z 427.007,A -85,B 0,C 180,E1 -26448.77,E2 -26448.77} C_VEL
LIN {X 0,Y 108.455,Z 426.976,A -85,B 0,C 180,E1 -26456.284,E2 -26456.284} C_VEL
LIN {X 0,Y 108.953,Z 426.914,A -85,B 0,C 180,E1 -26460,E2 -26460} C_VEL
LIN {X 0,Y 108.338,Z 426.939,A -85,B 0,C 180,E1 -26467.454,E2 -26467.454} C_VEL
LIN {X 0,Y 108.188,Z 427.007,A -85,B 0,C 180,E1 -26473.22,E2 -26473.22} C_VEL
LIN {X 0,Y 107.919,Z 426.995,A -85,B 0,C 180,E1 -26479.003,E2 -26479.003} C_VEL
LIN {X 0,Y 107.867,Z 427.031,A -85,B 0,C 180,E1 -26484.179,E2 -26484.179} C_VEL
LIN {X 0,Y 107.708,Z 427.038,A -85,B 0,C 180,E1 -26489.355,E2 -26489.355} C_VEL
LIN {X 0,Y 107.053,Z 427.33,A -85,B 0,C 180,E1 -26491.47,E2 -26491.47} C_VEL
LIN {X 0,Y 104.451,Z 428.799,A -85,B 0,C 180,E1 -26494.822,E2 -26494.822} C_VEL
LIN {X 0,Y 102.532,Z 430.951,A -85,B 0,C 180,E1 -26498.23,E2 -26498.23} C_VEL
LIN {X 0,Y 102.946,Z 432.324,A -85,B 0,C 180,E1 -26500.296,E2 -26500.296} C_VEL
LIN {X 0,Y 104.643,Z 433.651,A -85,B 0,C 180,E1 -26502.586,E2 -26502.586} C_VEL
LIN {X 0,Y 106.031,Z 436.582,A -85,B 0,C 180,E1 -26504.913,E2 -26504.913} C_VEL
LIN {X 0,Y 107.968,Z 438.644,A -85,B 0,C 180,E1 -26507.284,E2 -26507.284} C_VEL
LIN {X 0,Y 109.982,Z 442.227,A -85,B 0,C 180,E1 -26510.069,E2 -26510.069} C_VEL
LIN {X 0,Y 113.952,Z 449.29,A -85,B 0,C 180,E1 -26515.15,E2 -26515.15} C_VEL
LIN {X 0,Y 117.079,Z 456.145,A -85,B 0,C 180,E1 -26519.402,E2 -26519.402} C_VEL
LIN {X 0,Y 120.113,Z 464.29,A -85,B 0,C 180,E1 -26523.997,E2 -26523.997} C_VEL
LIN {X 0,Y 121.754,Z 470.915,A -85,B 0,C 180,E1 -26527.453,E2 -26527.453} C_VEL
LIN {X 0,Y 121.866,Z 474.834,A -85,B 0,C 180,E1 -26529.249,E2 -26529.249} C_VEL
LIN {X 0,Y 121.546,Z 479.756,A -85,B 0,C 180,E1 -26531.479,E2 -26531.479} C_VEL
LIN {X 0,Y 118.897,Z 485.726,A -85,B 0,C 180,E1 -26533.687,E2 -26533.687} C_VEL
LIN {X 0,Y 114.506,Z 494.075,A -85,B 0,C 180,E1 -26537.408,E2 -26537.408} C_VEL
LIN {X 0,Y 109.498,Z 502.854,A -85,B 0,C 180,E1 -26542.618,E2 -26542.618} C_VEL
LIN {X 0,Y 105.473,Z 509.735,A -85,B 0,C 180,E1 -26548.182,E2 -26548.182} C_VEL
LIN {X 0,Y 102.405,Z 514.989,A -85,B 0,C 180,E1 -26553.928,E2 -26553.928} C_VEL
LIN {X 0,Y 100.025,Z 519.295,A -85,B 0,C 180,E1 -26560.368,E2 -26560.368} C_VEL
LIN {X 0,Y 98.617,Z 522.213,A -85,B 0,C 180,E1 -26566.554,E2 -26566.554} C_VEL
LIN {X 0,Y 98.235,Z 523.838,A -85,B 0,C 180,E1 -26571.557,E2 -26571.557} C_VEL
LIN {X 0,Y 98.314,Z 524.673,A -85,B 0,C 180,E1 -26575.389,E2 -26575.389} C_VEL
LIN {X 0,Y 99.308,Z 525.301,A -85,B 0,C 180,E1 -26581.871,E2 -26581.871} C_VEL
LIN {X 0,Y 101.433,Z 524.896,A -85,B 0,C 180,E1 -26588.568,E2 -26588.568} C_VEL
LIN {X 0,Y 103.413,Z 524.013,A -85,B 0,C 180,E1 -26592.802,E2 -26592.802} C_VEL
LIN {X 0,Y 107.602,Z 521.62,A -85,B 0,C 180,E1 -26599.221,E2 -26599.221} C_VEL
LIN {X 0,Y 112.183,Z 518.401,A -85,B 0,C 180,E1 -26604.517,E2 -26604.517} C_VEL
LIN {X 0,Y 118.042,Z 513.711,A -85,B 0,C 180,E1 -26609.674,E2 -26609.674} C_VEL
LIN {X 0,Y 124.73,Z 507.524,A -85,B 0,C 180,E1 -26614.344,E2 -26614.344} C_VEL
LIN {X 0,Y 130.862,Z 500.998,A -85,B 0,C 180,E1 -26617.918,E2 -26617.918} C_VEL
LIN {X 0,Y 134.723,Z 496.458,A -85,B 0,C 180,E1 -26619.864,E2 -26619.864} C_VEL
LIN {X 0,Y 135.528,Z 494.968,A -85,B 0,C 180,E1 -26620.746,E2 -26620.746} C_VEL
LIN {X 0,Y 136.484,Z 491.205,A -85,B 0,C 180,E1 -26623.548,E2 -26623.548} C_VEL
LIN {X 0,Y 136.758,Z 487.564,A -85,B 0,C 180,E1 -26626.781,E2 -26626.781} C_VEL
LIN {X 0,Y 136.631,Z 483.338,A -85,B 0,C 180,E1 -26631.123,E2 -26631.123} C_VEL
LIN {X 0,Y 136.487,Z 480.896,A -85,B 0,C 180,E1 -26634.089,E2 -26634.089} C_VEL
LIN {X 0,Y 135.893,Z 477.418,A -85,B 0,C 180,E1 -26640,E2 -26640} C_VEL
LIN {X 0,Y 135.837,Z 476.003,A -85,B 0,C 180,E1 -26642.966,E2 -26642.966} C_VEL
LIN {X 0,Y 135.013,Z 475.934,A -85,B 0,C 180,E1 -26648.54,E2 -26648.54} C_VEL
LIN {X 0,Y 134.826,Z 476.474,A -85,B 0,C 180,E1 -26652.035,E2 -26652.035} C_VEL
LIN {X 0,Y 134.88,Z 477.29,A -85,B 0,C 180,E1 -26655.102,E2 -26655.102} C_VEL
LIN {X 0,Y 134.962,Z 478.729,A -85,B 0,C 180,E1 -26658.207,E2 -26658.207} C_VEL
LIN {X 0,Y 135.13,Z 481.925,A -85,B 0,C 180,E1 -26662.959,E2 -26662.959} C_VEL
LIN {X 0,Y 135.357,Z 486.618,A -85,B 0,C 180,E1 -26668.048,E2 -26668.048} C_VEL
LIN {X 0,Y 135.394,Z 492.344,A -85,B 0,C 180,E1 -26673.053,E2 -26673.053} C_VEL
LIN {X 0,Y 135.223,Z 495.89,A -85,B 0,C 180,E1 -26675.782,E2 -26675.782} C_VEL
LIN {X 0,Y 132.718,Z 501.463,A -85,B 0,C 180,E1 -26678.62,E2 -26678.62} C_VEL
LIN {X 0,Y 128.585,Z 508.756,A -85,B 0,C 180,E1 -26682.461,E2 -26682.461} C_VEL
LIN {X 0,Y 124.988,Z 513.815,A -85,B 0,C 180,E1 -26685.353,E2 -26685.353} C_VEL
LIN {X 0,Y 118.628,Z 520.296,A -85,B 0,C 180,E1 -26689.341,E2 -26689.341} C_VEL
LIN {X 0,Y 112.418,Z 526.064,A -85,B 0,C 180,E1 -26694.363,E2 -26694.363} C_VEL
LIN {X 0,Y 106.792,Z 530.787,A -85,B 0,C 180,E1 -26700.433,E2 -26700.433} C_VEL
LIN {X 0,Y 103.132,Z 533.612,A -85,B 0,C 180,E1 -26705.875,E2 -26705.875} C_VEL
LIN {X 0,Y 99.833,Z 535.99,A -85,B 0,C 180,E1 -26713.653,E2 -26713.653} C_VEL
LIN {X 0,Y 98.919,Z 536.608,A -85,B 0,C 180,E1 -26717.702,E2 -26717.702} C_VEL
LIN {X 0,Y 98.465,Z 536.816,A -85,B 0,C 180,E1 -26721.801,E2 -26721.801} C_VEL
LIN {X 0,Y 98.453,Z 536.425,A -85,B 0,C 180,E1 -26728.005,E2 -26728.005} C_VEL
LIN {X 0,Y 98.604,Z 536.081,A -85,B 0,C 180,E1 -26730.008,E2 -26730.008} C_VEL
LIN {X 0,Y 98.448,Z 535.071,A -85,B 0,C 180,E1 -26734.101,E2 -26734.101} C_VEL
LIN {X 0,Y 98.55,Z 533.591,A -85,B 0,C 180,E1 -26738.208,E2 -26738.208} C_VEL
LIN {X 0,Y 99.457,Z 530.558,A -85,B 0,C 180,E1 -26744.327,E2 -26744.327} C_VEL
LIN {X 0,Y 101.262,Z 526.436,A -85,B 0,C 180,E1 -26750.313,E2 -26750.313} C_VEL
LIN {X 0,Y 104.749,Z 520.123,A -85,B 0,C 180,E1 -26756.936,E2 -26756.936} C_VEL
LIN {X 0,Y 108.488,Z 513.405,A -85,B 0,C 180,E1 -26762.145,E2 -26762.145} C_VEL
LIN {X 0,Y 112.644,Z 506.188,A -85,B 0,C 180,E1 -26766.358,E2 -26766.358} C_VEL
LIN {X 0,Y 114.29,Z 502.95,A -85,B 0,C 180,E1 -26767.954,E2 -26767.954} C_VEL
LIN {X 0,Y 116.267,Z 495.284,A -85,B 0,C 180,E1 -26771.684,E2 -26771.684} C_VEL
LIN {X 0,Y 118.207,Z 484.798,A -85,B 0,C 180,E1 -26776.07,E2 -26776.07} C_VEL
LIN {X 0,Y 119.255,Z 475.149,A -85,B 0,C 180,E1 -26779.589,E2 -26779.589} C_VEL
LIN {X 0,Y 119.258,Z 470.986,A -85,B 0,C 180,E1 -26781.1,E2 -26781.1} C_VEL
LIN {X 0,Y 117.52,Z 463.9,A -85,B 0,C 180,E1 -26784.332,E2 -26784.332} C_VEL
LIN {X 0,Y 114.623,Z 455.162,A -85,B 0,C 180,E1 -26788.591,E2 -26788.591} C_VEL
LIN {X 0,Y 110.862,Z 446.008,A -85,B 0,C 180,E1 -26793.656,E2 -26793.656} C_VEL
LIN {X 0,Y 108.739,Z 441.734,A -85,B 0,C 180,E1 -26796.427,E2 -26796.427} C_VEL
LIN {X 0,Y 108.014,Z 440.237,A -85,B 0,C 180,E1 -26797.4,E2 -26797.4} C_VEL
LIN {X 0,Y 105.887,Z 436.634,A -85,B 0,C 180,E1 -26800.239,E2 -26800.239} C_VEL
LIN {X 0,Y 105.151,Z 434.629,A -85,B 0,C 180,E1 -26801.489,E2 -26801.489} C_VEL
LIN {X 0,Y 102.571,Z 431.578,A -85,B 0,C 180,E1 -26805.074,E2 -26805.074} C_VEL
LIN {X 0,Y 101.396,Z 429.054,A -85,B 0,C 180,E1 -26807.237,E2 -26807.237} C_VEL
LIN {X 0,Y 101.166,Z 427.891,A -85,B 0,C 180,E1 -26807.97,E2 -26807.97} C_VEL
LIN {X 0,Y 101.252,Z 427.877,A -85,B 0,C 180,E1 -26812.02,E2 -26812.02} C_VEL
LIN {X 0,Y 101.876,Z 427.795,A -85,B 0,C 180,E1 -26820,E2 -26820} C_VEL
LIN {X 0,Y 101.277,Z 427.819,A -85,B 0,C 180,E1 -26827.977,E2 -26827.977} C_VEL
LIN {X 0,Y 101.136,Z 427.887,A -85,B 0,C 180,E1 -26833.349,E2 -26833.349} C_VEL
LIN {X 0,Y 100.829,Z 427.874,A -85,B 0,C 180,E1 -26840.396,E2 -26840.396} C_VEL
LIN {X 0,Y 100.785,Z 427.922,A -85,B 0,C 180,E1 -26844.955,E2 -26844.955} C_VEL
LIN {X 0,Y 100.698,Z 427.896,A -85,B 0,C 180,E1 -26853.11,E2 -26853.11} C_VEL
LIN {X 0,Y 100.702,Z 428.064,A -85,B 0,C 180,E1 -26856.075,E2 -26856.075} C_VEL
LIN {X 0,Y 101.357,Z 430.268,A -85,B 0,C 180,E1 -26857.665,E2 -26857.665} C_VEL
LIN {X 0,Y 102.946,Z 432.324,A -85,B 0,C 180,E1 -26860.296,E2 -26860.296} C_VEL
LIN {X 0,Y 104.134,Z 433.982,A -85,B 0,C 180,E1 -26862.147,E2 -26862.147} C_VEL
LIN {X 0,Y 105.447,Z 437.501,A -85,B 0,C 180,E1 -26864.644,E2 -26864.644} C_VEL
LIN {X 0,Y 106.32,Z 441.687,A -85,B 0,C 180,E1 -26866.897,E2 -26866.897} C_VEL
LIN {X 0,Y 107.876,Z 450.418,A -85,B 0,C 180,E1 -26871.413,E2 -26871.413} C_VEL
LIN {X 0,Y 108.741,Z 452.896,A -85,B 0,C 180,E1 -26873.053,E2 -26873.053} C_VEL
LIN {X 0,Y 111.244,Z 458.601,A -85,B 0,C 180,E1 -26877.017,E2 -26877.017} C_VEL
LIN {X 0,Y 114.223,Z 467.045,A -85,B 0,C 180,E1 -26882.349,E2 -26882.349} C_VEL
LIN {X 0,Y 115.761,Z 473.836,A -85,B 0,C 180,E1 -26886.249,E2 -26886.249} C_VEL
LIN {X 0,Y 115.743,Z 477.646,A -85,B 0,C 180,E1 -26888.134,E2 -26888.134} C_VEL
LIN {X 0,Y 115.44,Z 480.464,A -85,B 0,C 180,E1 -26889.502,E2 -26889.502} C_VEL
LIN {X 0,Y 114.37,Z 483.398,A -85,B 0,C 180,E1 -26890.707,E2 -26890.707} C_VEL
LIN {X 0,Y 108.966,Z 493.416,A -85,B 0,C 180,E1 -26895.042,E2 -26895.042} C_VEL
LIN {X 0,Y 103.742,Z 502.133,A -85,B 0,C 180,E1 -26900.242,E2 -26900.242} C_VEL
LIN {X 0,Y 99.418,Z 509.118,A -85,B 0,C 180,E1 -26905.939,E2 -26905.939} C_VEL
LIN {X 0,Y 95.913,Z 514.703,A -85,B 0,C 180,E1 -26912.092,E2 -26912.092} C_VEL
LIN {X 0,Y 93.343,Z 519.049,A -85,B 0,C 180,E1 -26918.652,E2 -26918.652} C_VEL
LIN {X 0,Y 92.1,Z 521.299,A -85,B 0,C 180,E1 -26923.225,E2 -26923.225} C_VEL
LIN {X 0,Y 91.352,Z 523.093,A -85,B 0,C 180,E1 -26927.913,E2 -26927.913} C_VEL
LIN {X 0,Y 91.122,Z 524.437,A -85,B 0,C 180,E1 -26932.673,E2 -26932.673} C_VEL
LIN {X 0,Y 91.432,Z 525.28,A -85,B 0,C 180,E1 -26937.454,E2 -26937.454} C_VEL
LIN {X 0,Y 92.498,Z 525.748,A -85,B 0,C 180,E1 -26943.303,E2 -26943.303} C_VEL
LIN {X 0,Y 95.421,Z 525.133,A -85,B 0,C 180,E1 -26951.508,E2 -26951.508} C_VEL
LIN {X 0,Y 97.787,Z 524.154,A -85,B 0,C 180,E1 -26955.935,E2 -26955.935} C_VEL
LIN {X 0,Y 101.784,Z 522.026,A -85,B 0,C 180,E1 -26961.579,E2 -26961.579} C_VEL
LIN {X 0,Y 107.786,Z 518.139,A -85,B 0,C 180,E1 -26967.941,E2 -26967.941} C_VEL
LIN {X 0,Y 114.253,Z 513.182,A -85,B 0,C 180,E1 -26973.1,E2 -26973.1} C_VEL
LIN {X 0,Y 121.502,Z 506.723,A -85,B 0,C 180,E1 -26977.722,E2 -26977.722} C_VEL
LIN {X 0,Y 128.062,Z 499.971,A -85,B 0,C 180,E1 -26981.177,E2 -26981.177} C_VEL
LIN {X 0,Y 129.355,Z 498.527,A -85,B 0,C 180,E1 -26981.797,E2 -26981.797} C_VEL
LIN {X 0,Y 130.178,Z 497.077,A -85,B 0,C 180,E1 -26982.727,E2 -26982.727} C_VEL
LIN {X 0,Y 130.975,Z 494.472,A -85,B 0,C 180,E1 -26984.959,E2 -26984.959} C_VEL
LIN {X 0,Y 131.401,Z 491.761,A -85,B 0,C 180,E1 -26987.647,E2 -26987.647} C_VEL
LIN {X 0,Y 131.632,Z 487.688,A -85,B 0,C 180,E1 -26992.33,E2 -26992.33} C_VEL
LIN {X 0,Y 131.659,Z 486.517,A -85,B 0,C 180,E1 -26993.872,E2 -26993.872} C_VEL
LIN {X 0,Y 131.534,Z 484.608,A -85,B 0,C 180,E1 -26996.937,E2 -26996.937} C_VEL
LIN {X 0,Y 131.537,Z 481.734,A -85,B 0,C 180,E1 -27003.063,E2 -27003.063} C_VEL
LIN {X 0,Y 131.103,Z 481.543,A -85,B 0,C 180,E1 -27006.155,E2 -27006.155} C_VEL
LIN {X 0,Y 130.761,Z 481.755,A -85,B 0,C 180,E1 -27009.279,E2 -27009.279} C_VEL
LIN {X 0,Y 130.624,Z 482.845,A -85,B 0,C 180,E1 -27014.456,E2 -27014.456} C_VEL
LIN {X 0,Y 130.467,Z 485.733,A -85,B 0,C 180,E1 -27020.168,E2 -27020.168} C_VEL
LIN {X 0,Y 130.465,Z 488.192,A -85,B 0,C 180,E1 -27023.703,E2 -27023.703} C_VEL
LIN {X 0,Y 130.297,Z 492.097,A -85,B 0,C 180,E1 -27028.03,E2 -27028.03} C_VEL
LIN {X 0,Y 129.943,Z 497.123,A -85,B 0,C 180,E1 -27032.742,E2 -27032.742} C_VEL
LIN {X 0,Y 129.8,Z 498.66,A -85,B 0,C 180,E1 -27034.051,E2 -27034.051} C_VEL
LIN {X 0,Y 128.131,Z 502.065,A -85,B 0,C 180,E1 -27036.006,E2 -27036.006} C_VEL
LIN {X 0,Y 123.766,Z 509.105,A -85,B 0,C 180,E1 -27039.962,E2 -27039.962} C_VEL
LIN {X 0,Y 119.988,Z 514.08,A -85,B 0,C 180,E1 -27042.943,E2 -27042.943} C_VEL
LIN {X 0,Y 113.336,Z 520.405,A -85,B 0,C 180,E1 -27047.001,E2 -27047.001} C_VEL
LIN {X 0,Y 106.248,Z 526.383,A -85,B 0,C 180,E1 -27052.539,E2 -27052.539} C_VEL
LIN {X 0,Y 100.656,Z 530.633,A -85,B 0,C 180,E1 -27058.431,E2 -27058.431} C_VEL
LIN {X 0,Y 96.655,Z 533.366,A -85,B 0,C 180,E1 -27064.143,E2 -27064.143} C_VEL
LIN {X 0,Y 92.999,Z 535.653,A -85,B 0,C 180,E1 -27072.414,E2 -27072.414} C_VEL
LIN {X 0,Y 91.411,Z 536.357,A -85,B 0,C 180,E1 -27081.163,E2 -27081.163} C_VEL
LIN {X 0,Y 91.397,Z 535.79,A -85,B 0,C 180,E1 -27088.473,E2 -27088.473} C_VEL
LIN {X 0,Y 91.433,Z 535.047,A -85,B 0,C 180,E1 -27092.209,E2 -27092.209} C_VEL
LIN {X 0,Y 91.525,Z 532.934,A -85,B 0,C 180,E1 -27098.843,E2 -27098.843} C_VEL
LIN {X 0,Y 92.578,Z 529.813,A -85,B 0,C 180,E1 -27105.417,E2 -27105.417} C_VEL
LIN {X 0,Y 94.601,Z 525.596,A -85,B 0,C 180,E1 -27111.814,E2 -27111.814} C_VEL
LIN {X 0,Y 97.816,Z 520.198,A -85,B 0,C 180,E1 -27117.849,E2 -27117.849} C_VEL
LIN {X 0,Y 101.863,Z 513.402,A -85,B 0,C 180,E1 -27123.51,E2 -27123.51} C_VEL
LIN {X 0,Y 106.97,Z 504.985,A -85,B 0,C 180,E1 -27128.629,E2 -27128.629} C_VEL
LIN {X 0,Y 108.427,Z 501.622,A -85,B 0,C 180,E1 -27130.413,E2 -27130.413} C_VEL
LIN {X 0,Y 110.737,Z 492.642,A -85,B 0,C 180,E1 -27134.899,E2 -27134.899} C_VEL
LIN {X 0,Y 112.465,Z 484.026,A -85,B 0,C 180,E1 -27138.59,E2 -27138.59} C_VEL
LIN {X 0,Y 113.496,Z 475.9,A -85,B 0,C 180,E1 -27141.74,E2 -27141.74} C_VEL
LIN {X 0,Y 113.391,Z 473.17,A -85,B 0,C 180,E1 -27142.921,E2 -27142.921} C_VEL
LIN {X 0,Y 111.723,Z 465.867,A -85,B 0,C 180,E1 -27146.603,E2 -27146.603} C_VEL
LIN {X 0,Y 109.215,Z 457.856,A -85,B 0,C 180,E1 -27151.045,E2 -27151.045} C_VEL
LIN {X 0,Y 106.379,Z 450.511,A -85,B 0,C 180,E1 -27155.612,E2 -27155.612} C_VEL
LIN {X 0,Y 104.779,Z 446.393,A -85,B 0,C 180,E1 -27158.351,E2 -27158.351} C_VEL
LIN {X 0,Y 102.543,Z 442.066,A -85,B 0,C 180,E1 -27161.947,E2 -27161.947} C_VEL
LIN {X 0,Y 101.896,Z 440.433,A -85,B 0,C 180,E1 -27163.212,E2 -27163.212} C_VEL
LIN {X 0,Y 99.44,Z 436.793,A -85,B 0,C 180,E1 -27167.402,E2 -27167.402} C_VEL
LIN {X 0,Y 98.601,Z 434.508,A -85,B 0,C 180,E1 -27169.476,E2 -27169.476} C_VEL
LIN {X 0,Y 95.898,Z 432.446,A -85,B 0,C 180,E1 -27175.007,E2 -27175.007} C_VEL
LIN {X 0,Y 94.899,Z 430.059,A -85,B 0,C 180,E1 -27178.541,E2 -27178.541} C_VEL
LIN {X 0,Y 94.792,Z 428.677,A -85,B 0,C 180,E1 -27179.867,E2 -27179.867} C_VEL
LIN {X 0,Y 94.21,Z 428.7,A -85,B 0,C 180,E1 -27188.58,E2 -27188.58} C_VEL
LIN {X 0,Y 94.054,Z 428.77,A -85,B 0,C 180,E1 -27193.706,E2 -27193.706} C_VEL
LIN {X 0,Y 93.767,Z 428.957,A -85,B 0,C 180,E1 -27201.576,E2 -27201.576} C_VEL
LIN {X 0,Y 94.973,Z 432.194,A -85,B 0,C 180,E1 -27207.546,E2 -27207.546} C_VEL
LIN {X 0,Y 98.103,Z 434.693,A -85,B 0,C 180,E1 -27214.751,E2 -27214.751} C_VEL
LIN {X 0,Y 99.234,Z 437.504,A -85,B 0,C 180,E1 -27217.65,E2 -27217.65} C_VEL
LIN {X 0,Y 101.732,Z 440.461,A -85,B 0,C 180,E1 -27221.88,E2 -27221.88} C_VEL
LIN {X 0,Y 103.383,Z 443.394,A -85,B 0,C 180,E1 -27224.822,E2 -27224.822} C_VEL
LIN {X 0,Y 104.301,Z 444.324,A -85,B 0,C 180,E1 -27226.05,E2 -27226.05} C_VEL
LIN {X 0,Y 107.73,Z 450.945,A -85,B 0,C 180,E1 -27231.522,E2 -27231.522} C_VEL
LIN {X 0,Y 108.741,Z 452.896,A -85,B 0,C 180,E1 -27233.053,E2 -27233.053} C_VEL
LIN {X 0,Y 109.602,Z 455.323,A -85,B 0,C 180,E1 -27234.618,E2 -27234.618} C_VEL
LIN {X 0,Y 110.189,Z 459.551,A -85,B 0,C 180,E1 -27236.766,E2 -27236.766} C_VEL
LIN {X 0,Y 110.14,Z 464.111,A -85,B 0,C 180,E1 -27238.768,E2 -27238.768} C_VEL
LIN {X 0,Y 109.522,Z 473.251,A -85,B 0,C 180,E1 -27242.947,E2 -27242.947} C_VEL
LIN {X 0,Y 109.651,Z 475.982,A -85,B 0,C 180,E1 -27244.503,E2 -27244.503} C_VEL
LIN {X 0,Y 109.865,Z 477.908,A -85,B 0,C 180,E1 -27245.651,E2 -27245.651} C_VEL
LIN {X 0,Y 109.049,Z 482.982,A -85,B 0,C 180,E1 -27248.242,E2 -27248.242} C_VEL
LIN {X 0,Y 104.26,Z 491.618,A -85,B 0,C 180,E1 -27251.942,E2 -27251.942} C_VEL
LIN {X 0,Y 99.073,Z 499.965,A -85,B 0,C 180,E1 -27256.663,E2 -27256.663} C_VEL
LIN {X 0,Y 94.147,Z 507.501,A -85,B 0,C 180,E1 -27262.486,E2 -27262.486} C_VEL
LIN {X 0,Y 90.648,Z 512.68,A -85,B 0,C 180,E1 -27267.882,E2 -27267.882} C_VEL
LIN {X 0,Y 87.489,Z 517.517,A -85,B 0,C 180,E1 -27274.599,E2 -27274.599} C_VEL
LIN {X 0,Y 85.681,Z 520.482,A -85,B 0,C 180,E1 -27280.166,E2 -27280.166} C_VEL
LIN {X 0,Y 84.736,Z 522.27,A -85,B 0,C 180,E1 -27284.398,E2 -27284.398} C_VEL
LIN {X 0,Y 84.041,Z 524.839,A -85,B 0,C 180,E1 -27293.092,E2 -27293.092} C_VEL
LIN {X 0,Y 84.635,Z 525.89,A -85,B 0,C 180,E1 -27299.872,E2 -27299.872} C_VEL
LIN {X 0,Y 85.751,Z 526.193,A -85,B 0,C 180,E1 -27304.997,E2 -27304.997} C_VEL
LIN {X 0,Y 87.441,Z 526.003,A -85,B 0,C 180,E1 -27310.003,E2 -27310.003} C_VEL
LIN {X 0,Y 89.905,Z 525.307,A -85,B 0,C 180,E1 -27315.289,E2 -27315.289} C_VEL
LIN {X 0,Y 92.478,Z 524.263,A -85,B 0,C 180,E1 -27319.447,E2 -27319.447} C_VEL
LIN {X 0,Y 96.185,Z 522.441,A -85,B 0,C 180,E1 -27324.23,E2 -27324.23} C_VEL
LIN {X 0,Y 101.628,Z 519.23,A -85,B 0,C 180,E1 -27329.8,E2 -27329.8} C_VEL
LIN {X 0,Y 108.449,Z 514.536,A -85,B 0,C 180,E1 -27335.111,E2 -27335.111} C_VEL
LIN {X 0,Y 116.041,Z 508.337,A -85,B 0,C 180,E1 -27339.82,E2 -27339.82} C_VEL
LIN {X 0,Y 124.304,Z 500.411,A -85,B 0,C 180,E1 -27343.952,E2 -27343.952} C_VEL
LIN {X 0,Y 125.098,Z 498.87,A -85,B 0,C 180,E1 -27345.245,E2 -27345.245} C_VEL
LIN {X 0,Y 125.676,Z 497.069,A -85,B 0,C 180,E1 -27347.075,E2 -27347.075} C_VEL
LIN {X 0,Y 126.37,Z 493.071,A -85,B 0,C 180,E1 -27352.008,E2 -27352.008} C_VEL
LIN {X 0,Y 126.529,Z 491.876,A -85,B 0,C 180,E1 -27353.622,E2 -27353.622} C_VEL
LIN {X 0,Y 126.65,Z 489.843,A -85,B 0,C 180,E1 -27357.096,E2 -27357.096} C_VEL
LIN {X 0,Y 126.909,Z 487.197,A -85,B 0,C 180,E1 -27363.175,E2 -27363.175} C_VEL
LIN {X 0,Y 126.553,Z 487.06,A -85,B 0,C 180,E1 -27366.377,E2 -27366.377} C_VEL
LIN {X 0,Y 126.218,Z 487.337,A -85,B 0,C 180,E1 -27369.616,E2 -27369.616} C_VEL
LIN {X 0,Y 126.076,Z 487.957,A -85,B 0,C 180,E1 -27372.884,E2 -27372.884} C_VEL
LIN {X 0,Y 125.805,Z 490.059,A -85,B 0,C 180,E1 -27378.274,E2 -27378.274} C_VEL
LIN {X 0,Y 125.658,Z 491.832,A -85,B 0,C 180,E1 -27381.318,E2 -27381.318} C_VEL
LIN {X 0,Y 125.104,Z 496.084,A -85,B 0,C 180,E1 -27386.707,E2 -27386.707} C_VEL
LIN {X 0,Y 124.314,Z 501.215,A -85,B 0,C 180,E1 -27392.017,E2 -27392.017} C_VEL
LIN {X 0,Y 123.813,Z 502.677,A -85,B 0,C 180,E1 -27393.164,E2 -27393.164} C_VEL
LIN {X 0,Y 120.097,Z 508.201,A -85,B 0,C 180,E1 -27396.437,E2 -27396.437} C_VEL
LIN {X 0,Y 115.199,Z 514.306,A -85,B 0,C 180,E1 -27400.318,E2 -27400.318} C_VEL
LIN {X 0,Y 110.555,Z 518.559,A -85,B 0,C 180,E1 -27403.036,E2 -27403.036} C_VEL
LIN {X 0,Y 103.858,Z 523.939,A -85,B 0,C 180,E1 -27407.426,E2 -27407.426} C_VEL
LIN {X 0,Y 98.123,Z 528.204,A -85,B 0,C 180,E1 -27412.508,E2 -27412.508} C_VEL
LIN {X 0,Y 93.07,Z 531.466,A -85,B 0,C 180,E1 -27418.1,E2 -27418.1} C_VEL
LIN {X 0,Y 87.941,Z 534.414,A -85,B 0,C 180,E1 -27426.458,E2 -27426.458} C_VEL
LIN {X 0,Y 85.04,Z 535.779,A -85,B 0,C 180,E1 -27435.655,E2 -27435.655} C_VEL
LIN {X 0,Y 84.208,Z 535.647,A -85,B 0,C 180,E1 -27445.222,E2 -27445.222} C_VEL
LIN {X 0,Y 84.446,Z 535,A -85,B 0,C 180,E1 -27450.009,E2 -27450.009} C_VEL
LIN {X 0,Y 84.294,Z 533.844,A -85,B 0,C 180,E1 -27454.792,E2 -27454.792} C_VEL
LIN {X 0,Y 84.771,Z 531.317,A -85,B 0,C 180,E1 -27461.971,E2 -27461.971} C_VEL
LIN {X 0,Y 86.333,Z 527.747,A -85,B 0,C 180,E1 -27469.012,E2 -27469.012} C_VEL
LIN {X 0,Y 89.135,Z 523.057,A -85,B 0,C 180,E1 -27475.709,E2 -27475.709} C_VEL
LIN {X 0,Y 93.69,Z 515.964,A -85,B 0,C 180,E1 -27482.955,E2 -27482.955} C_VEL
LIN {X 0,Y 97.823,Z 509.486,A -85,B 0,C 180,E1 -27487.787,E2 -27487.787} C_VEL
LIN {X 0,Y 101.452,Z 503.677,A -85,B 0,C 180,E1 -27491.164,E2 -27491.164} C_VEL
LIN {X 0,Y 103.84,Z 496.284,A -85,B 0,C 180,E1 -27495.297,E2 -27495.297} C_VEL
LIN {X 0,Y 106.368,Z 485.913,A -85,B 0,C 180,E1 -27500.231,E2 -27500.231} C_VEL
LIN {X 0,Y 107.698,Z 478.284,A -85,B 0,C 180,E1 -27503.454,E2 -27503.454} C_VEL
LIN {X 0,Y 107.475,Z 474.97,A -85,B 0,C 180,E1 -27505.097,E2 -27505.097} C_VEL
LIN {X 0,Y 105.699,Z 466.68,A -85,B 0,C 180,E1 -27509.824,E2 -27509.824} C_VEL
LIN {X 0,Y 103.336,Z 458.804,A -85,B 0,C 180,E1 -27514.845,E2 -27514.845} C_VEL
LIN {X 0,Y 100.525,Z 450.993,A -85,B 0,C 180,E1 -27520.604,E2 -27520.604} C_VEL
LIN {X 0,Y 98.156,Z 445.726,A -85,B 0,C 180,E1 -27525.487,E2 -27525.487} C_VEL
LIN {X 0,Y 96.088,Z 441.101,A -85,B 0,C 180,E1 -27530.527,E2 -27530.527} C_VEL
LIN {X 0,Y 93.622,Z 438.756,A -85,B 0,C 180,E1 -27536.503,E2 -27536.503} C_VEL
LIN {X 0,Y 92.838,Z 436.03,A -85,B 0,C 180,E1 -27540.542,E2 -27540.542} C_VEL
LIN {X 0,Y 92.806,Z 435.522,A -85,B 0,C 180,E1 -27541.084,E2 -27541.084} C_VEL
LIN {X 0,Y 91.185,Z 435.253,A -85,B 0,C 180,E1 -27553.369,E2 -27553.369} C_VEL
LIN {X 0,Y 91.908,Z 435.728,A -85,B 0,C 180,E1 -27560.565,E2 -27560.565} C_VEL
LIN {X 0,Y 93.218,Z 439.356,A -85,B 0,C 180,E1 -27568.185,E2 -27568.185} C_VEL
LIN {X 0,Y 95.275,Z 440.935,A -85,B 0,C 180,E1 -27573.293,E2 -27573.293} C_VEL
LIN {X 0,Y 96.304,Z 443.715,A -85,B 0,C 180,E1 -27576.594,E2 -27576.594} C_VEL
LIN {X 0,Y 98.581,Z 446.964,A -85,B 0,C 180,E1 -27581.258,E2 -27581.258} C_VEL
LIN {X 0,Y 100.947,Z 451.158,A -85,B 0,C 180,E1 -27585.867,E2 -27585.867} C_VEL
LIN {X 0,Y 103.787,Z 456.996,A -85,B 0,C 180,E1 -27591.147,E2 -27591.147} C_VEL
LIN {X 0,Y 105.891,Z 462.21,A -85,B 0,C 180,E1 -27595.23,E2 -27595.23} C_VEL
LIN {X 0,Y 108.006,Z 468.73,A -85,B 0,C 180,E1 -27599.773,E2 -27599.773} C_VEL
LIN {X 0,Y 109.517,Z 475.093,A -85,B 0,C 180,E1 -27603.951,E2 -27603.951} C_VEL
LIN {X 0,Y 109.651,Z 475.982,A -85,B 0,C 180,E1 -27604.503,E2 -27604.503} C_VEL
LIN {X 0,Y 109.274,Z 478.325,A -85,B 0,C 180,E1 -27605.605,E2 -27605.605} C_VEL
LIN {X 0,Y 107.205,Z 481.841,A -85,B 0,C 180,E1 -27606.687,E2 -27606.687} C_VEL
LIN {X 0,Y 100.058,Z 489.798,A -85,B 0,C 180,E1 -27608.672,E2 -27608.672} C_VEL
LIN {X 0,Y 98.612,Z 491.76,A -85,B 0,C 180,E1 -27609.52,E2 -27609.52} C_VEL
LIN {X 0,Y 92.865,Z 500.497,A -85,B 0,C 180,E1 -27614.632,E2 -27614.632} C_VEL
LIN {X 0,Y 87.607,Z 508.015,A -85,B 0,C 180,E1 -27620.759,E2 -27620.759} C_VEL
LIN {X 0,Y 83.295,Z 513.98,A -85,B 0,C 180,E1 -27627.573,E2 -27627.573} C_VEL
LIN {X 0,Y 80.054,Z 518.673,A -85,B 0,C 180,E1 -27635.027,E2 -27635.027} C_VEL
LIN {X 0,Y 77.845,Z 522.242,A -85,B 0,C 180,E1 -27643.034,E2 -27643.034} C_VEL
LIN {X 0,Y 76.987,Z 525.326,A -85,B 0,C 180,E1 -27654.094,E2 -27654.094} C_VEL
LIN {X 0,Y 78.011,Z 526.465,A -85,B 0,C 180,E1 -27662.708,E2 -27662.708} C_VEL
LIN {X 0,Y 79.482,Z 526.62,A -85,B 0,C 180,E1 -27668.227,E2 -27668.227} C_VEL
LIN {X 0,Y 81.576,Z 526.343,A -85,B 0,C 180,E1 -27673.554,E2 -27673.554} C_VEL
LIN {X 0,Y 84.275,Z 525.585,A -85,B 0,C 180,E1 -27678.623,E2 -27678.623} C_VEL
LIN {X 0,Y 87.564,Z 524.326,A -85,B 0,C 180,E1 -27683.364,E2 -27683.364} C_VEL
LIN {X 0,Y 93.413,Z 521.519,A -85,B 0,C 180,E1 -27689.889,E2 -27689.889} C_VEL
LIN {X 0,Y 100.279,Z 517.494,A -85,B 0,C 180,E1 -27695.637,E2 -27695.637} C_VEL
LIN {X 0,Y 107.203,Z 512.708,A -85,B 0,C 180,E1 -27700.127,E2 -27700.127} C_VEL
LIN {X 0,Y 114.982,Z 506.382,A -85,B 0,C 180,E1 -27704.269,E2 -27704.269} C_VEL
LIN {X 0,Y 119.272,Z 502.318,A -85,B 0,C 180,E1 -27706.368,E2 -27706.368} C_VEL
LIN {X 0,Y 120.026,Z 500.693,A -85,B 0,C 180,E1 -27708.174,E2 -27708.174} C_VEL
LIN {X 0,Y 121.064,Z 497.003,A -85,B 0,C 180,E1 -27713.333,E2 -27713.333} C_VEL
LIN {X 0,Y 121.393,Z 495.105,A -85,B 0,C 180,E1 -27716.681,E2 -27716.681} C_VEL
LIN {X 0,Y 121.667,Z 493.631,A -85,B 0,C 180,E1 -27720,E2 -27720} C_VEL
LIN {X 0,Y 121.998,Z 492.399,A -85,B 0,C 180,E1 -27723.303,E2 -27723.303} C_VEL
LIN {X 0,Y 121.693,Z 492.29,A -85,B 0,C 180,E1 -27726.633,E2 -27726.633} C_VEL
LIN {X 0,Y 121.337,Z 492.661,A -85,B 0,C 180,E1 -27730.092,E2 -27730.092} C_VEL
LIN {X 0,Y 121.137,Z 493.382,A -85,B 0,C 180,E1 -27733.419,E2 -27733.419} C_VEL
LIN {X 0,Y 120.878,Z 494.622,A -85,B 0,C 180,E1 -27736.901,E2 -27736.901} C_VEL
LIN {X 0,Y 120.497,Z 496.869,A -85,B 0,C 180,E1 -27741.081,E2 -27741.081} C_VEL
LIN {X 0,Y 119.669,Z 500.498,A -85,B 0,C 180,E1 -27746.063,E2 -27746.063} C_VEL
LIN {X 0,Y 118.824,Z 504.016,A -85,B 0,C 180,E1 -27750.132,E2 -27750.132} C_VEL
LIN {X 0,Y 118.28,Z 505.427,A -85,B 0,C 180,E1 -27751.458,E2 -27751.458} C_VEL
LIN {X 0,Y 113.676,Z 511.249,A -85,B 0,C 180,E1 -27755.195,E2 -27755.195} C_VEL
LIN {X 0,Y 109.533,Z 515.672,A -85,B 0,C 180,E1 -27758.2,E2 -27758.2} C_VEL
LIN {X 0,Y 101.019,Z 522.363,A -85,B 0,C 180,E1 -27763.085,E2 -27763.085} C_VEL
LIN {X 0,Y 93.276,Z 527.647,A -85,B 0,C 180,E1 -27769.11,E2 -27769.11} C_VEL
LIN {X 0,Y 87.093,Z 531.286,A -85,B 0,C 180,E1 -27775.618,E2 -27775.618} C_VEL
LIN {X 0,Y 84.041,Z 532.905,A -85,B 0,C 180,E1 -27779.895,E2 -27779.895} C_VEL
LIN {X 0,Y 81.444,Z 534.105,A -85,B 0,C 180,E1 -27784.451,E2 -27784.451} C_VEL
LIN {X 0,Y 78.152,Z 535.364,A -85,B 0,C 180,E1 -27794.359,E2 -27794.359} C_VEL
LIN {X 0,Y 77.134,Z 535.144,A -85,B 0,C 180,E1 -27804.782,E2 -27804.782} C_VEL
LIN {X 0,Y 77.325,Z 534.18,A -85,B 0,C 180,E1 -27811.181,E2 -27811.181} C_VEL
LIN {X 0,Y 77.475,Z 531.588,A -85,B 0,C 180,E1 -27820.463,E2 -27820.463} C_VEL
LIN {X 0,Y 78.881,Z 528.278,A -85,B 0,C 180,E1 -27828.18,E2 -27828.18} C_VEL
LIN {X 0,Y 81.536,Z 523.87,A -85,B 0,C 180,E1 -27835.539,E2 -27835.539} C_VEL
LIN {X 0,Y 85.429,Z 518.254,A -85,B 0,C 180,E1 -27842.336,E2 -27842.336} C_VEL
LIN {X 0,Y 89.379,Z 512.456,A -85,B 0,C 180,E1 -27847.555,E2 -27847.555} C_VEL
LIN {X 0,Y 95.166,Z 504.014,A -85,B 0,C 180,E1 -27853.097,E2 -27853.097} C_VEL
LIN {X 0,Y 97.793,Z 496.706,A -85,B 0,C 180,E1 -27857.455,E2 -27857.455} C_VEL
LIN {X 0,Y 100.634,Z 486.537,A -85,B 0,C 180,E1 -27862.609,E2 -27862.609} C_VEL
LIN {X 0,Y 101.957,Z 479.577,A -85,B 0,C 180,E1 -27865.821,E2 -27865.821} C_VEL
LIN {X 0,Y 100.74,Z 471.641,A -85,B 0,C 180,E1 -27870.768,E2 -27870.768} C_VEL
LIN {X 0,Y 98.968,Z 464.121,A -85,B 0,C 180,E1 -27875.9,E2 -27875.9} C_VEL
LIN {X 0,Y 96.69,Z 456.472,A -85,B 0,C 180,E1 -27882.005,E2 -27882.005} C_VEL
LIN {X 0,Y 95.498,Z 453.169,A -85,B 0,C 180,E1 -27885.073,E2 -27885.073} C_VEL
LIN {X 0,Y 93.306,Z 447.842,A -85,B 0,C 180,E1 -27891.335,E2 -27891.335} C_VEL
LIN {X 0,Y 91.099,Z 444.998,A -85,B 0,C 180,E1 -27897.927,E2 -27897.927} C_VEL
LIN {X 0,Y 90.552,Z 442.33,A -85,B 0,C 180,E1 -27902.224,E2 -27902.224} C_VEL
LIN {X 0,Y 89.245,Z 442.096,A -85,B 0,C 180,E1 -27913.665,E2 -27913.665} C_VEL
LIN {X 0,Y 89.76,Z 442.589,A -85,B 0,C 180,E1 -27919.998,E2 -27919.998} C_VEL
LIN {X 0,Y 90.754,Z 445.961,A -85,B 0,C 180,E1 -27927.687,E2 -27927.687} C_VEL
LIN {X 0,Y 92.307,Z 447.328,A -85,B 0,C 180,E1 -27932.205,E2 -27932.205} C_VEL
LIN {X 0,Y 93.665,Z 450.609,A -85,B 0,C 180,E1 -27936.889,E2 -27936.889} C_VEL
LIN {X 0,Y 94.617,Z 452,A -85,B 0,C 180,E1 -27939.15,E2 -27939.15} C_VEL
LIN {X 0,Y 96.869,Z 456.528,A -85,B 0,C 180,E1 -27944.591,E2 -27944.591} C_VEL
LIN {X 0,Y 99.384,Z 462.511,A -85,B 0,C 180,E1 -27950.464,E2 -27950.464} C_VEL
LIN {X 0,Y 101.087,Z 467.466,A -85,B 0,C 180,E1 -27954.635,E2 -27954.635} C_VEL
LIN {X 0,Y 103.076,Z 475.116,A -85,B 0,C 180,E1 -27960.435,E2 -27960.435} C_VEL
LIN {X 0,Y 103.827,Z 480.409,A -85,B 0,C 180,E1 -27964.109,E2 -27964.109} C_VEL
LIN {X 0,Y 103.275,Z 483.61,A -85,B 0,C 180,E1 -27965.894,E2 -27965.894} C_VEL
LIN {X 0,Y 98.612,Z 491.76,A -85,B 0,C 180,E1 -27969.52,E2 -27969.52} C_VEL
LIN {X 0,Y 95.569,Z 495.745,A -85,B 0,C 180,E1 -27971.408,E2 -27971.408} C_VEL
LIN {X 0,Y 89.14,Z 501.757,A -85,B 0,C 180,E1 -27974.248,E2 -27974.248} C_VEL
LIN {X 0,Y 82.704,Z 507.194,A -85,B 0,C 180,E1 -27977.744,E2 -27977.744} C_VEL
LIN {X 0,Y 79.786,Z 510.22,A -85,B 0,C 180,E1 -27980.661,E2 -27980.661} C_VEL
LIN {X 0,Y 75.853,Z 515.297,A -85,B 0,C 180,E1 -27987.335,E2 -27987.335} C_VEL
LIN {X 0,Y 72.564,Z 519.803,A -85,B 0,C 180,E1 -27995.547,E2 -27995.547} C_VEL
LIN {X 0,Y 70.999,Z 522.203,A -85,B 0,C 180,E1 -28001.407,E2 -28001.407} C_VEL
LIN {X 0,Y 70.05,Z 524.078,A -85,B 0,C 180,E1 -28007.505,E2 -28007.505} C_VEL
LIN {X 0,Y 69.963,Z 525.807,A -85,B 0,C 180,E1 -28015.301,E2 -28015.301} C_VEL
LIN {X 0,Y 71.603,Z 526.981,A -85,B 0,C 180,E1 -28026.066,E2 -28026.066} C_VEL
LIN {X 0,Y 73.504,Z 527.049,A -85,B 0,C 180,E1 -28031.998,E2 -28031.998} C_VEL
LIN {X 0,Y 77.968,Z 526.178,A -85,B 0,C 180,E1 -28040.878,E2 -28040.878} C_VEL
LIN {X 0,Y 83.091,Z 524.409,A -85,B 0,C 180,E1 -28047.741,E2 -28047.741} C_VEL
LIN {X 0,Y 89.695,Z 521.411,A -85,B 0,C 180,E1 -28054.277,E2 -28054.277} C_VEL
LIN {X 0,Y 97.301,Z 517.146,A -85,B 0,C 180,E1 -28059.855,E2 -28059.855} C_VEL
LIN {X 0,Y 106.696,Z 510.723,A -85,B 0,C 180,E1 -28065.168,E2 -28065.168} C_VEL
LIN {X 0,Y 113.3,Z 505.384,A -85,B 0,C 180,E1 -28068.195,E2 -28068.195} C_VEL
LIN {X 0,Y 114.36,Z 504.092,A -85,B 0,C 180,E1 -28069.465,E2 -28069.465} C_VEL
LIN {X 0,Y 115.266,Z 501.807,A -85,B 0,C 180,E1 -28072.996,E2 -28072.996} C_VEL
LIN {X 0,Y 115.858,Z 499.954,A -85,B 0,C 180,E1 -28076.523,E2 -28076.523} C_VEL
LIN {X 0,Y 116.34,Z 498.513,A -85,B 0,C 180,E1 -28080,E2 -28080} C_VEL
LIN {X 0,Y 116.834,Z 497.326,A -85,B 0,C 180,E1 -28083.449,E2 -28083.449} C_VEL
LIN {X 0,Y 116.535,Z 497.283,A -85,B 0,C 180,E1 -28086.928,E2 -28086.928} C_VEL
LIN {X 0,Y 116.183,Z 497.707,A -85,B 0,C 180,E1 -28090.456,E2 -28090.456} C_VEL
LIN {X 0,Y 115.894,Z 498.558,A -85,B 0,C 180,E1 -28094.038,E2 -28094.038} C_VEL
LIN {X 0,Y 115.467,Z 499.99,A -85,B 0,C 180,E1 -28097.718,E2 -28097.718} C_VEL
LIN {X 0,Y 114.937,Z 501.978,A -85,B 0,C 180,E1 -28101.524,E2 -28101.524} C_VEL
LIN {X 0,Y 113.979,Z 504.806,A -85,B 0,C 180,E1 -28105.571,E2 -28105.571} C_VEL
LIN {X 0,Y 112.868,Z 507.834,A -85,B 0,C 180,E1 -28109.354,E2 -28109.354} C_VEL
LIN {X 0,Y 110.363,Z 510.757,A -85,B 0,C 180,E1 -28111.42,E2 -28111.42} C_VEL
LIN {X 0,Y 105.221,Z 515.92,A -85,B 0,C 180,E1 -28115.108,E2 -28115.108} C_VEL
LIN {X 0,Y 98.813,Z 520.735,A -85,B 0,C 180,E1 -28118.536,E2 -28118.536} C_VEL
LIN {X 0,Y 91.566,Z 525.475,A -85,B 0,C 180,E1 -28123.198,E2 -28123.198} C_VEL
LIN {X 0,Y 85.182,Z 529.172,A -85,B 0,C 180,E1 -28128.71,E2 -28128.71} C_VEL
LIN {X 0,Y 81.31,Z 531.123,A -85,B 0,C 180,E1 -28132.781,E2 -28132.781} C_VEL
LIN {X 0,Y 77.956,Z 532.658,A -85,B 0,C 180,E1 -28137.266,E2 -28137.266} C_VEL
LIN {X 0,Y 72.884,Z 534.551,A -85,B 0,C 180,E1 -28147.324,E2 -28147.324} C_VEL
LIN {X 0,Y 70.394,Z 534.983,A -85,B 0,C 180,E1 -28158.493,E2 -28158.493} C_VEL
LIN {X 0,Y 70.057,Z 534.604,A -85,B 0,C 180,E1 -28164.254,E2 -28164.254} C_VEL
LIN {X 0,Y 70.281,Z 533.825,A -85,B 0,C 180,E1 -28170.011,E2 -28170.011} C_VEL
LIN {X 0,Y 70.143,Z 532.572,A -85,B 0,C 180,E1 -28175.761,E2 -28175.761} C_VEL
LIN {X 0,Y 70.914,Z 529.857,A -85,B 0,C 180,E1 -28184.356,E2 -28184.356} C_VEL
LIN {X 0,Y 72.993,Z 526.084,A -85,B 0,C 180,E1 -28192.663,E2 -28192.663} C_VEL
LIN {X 0,Y 76.499,Z 521.178,A -85,B 0,C 180,E1 -28200.362,E2 -28200.362} C_VEL
LIN {X 0,Y 81.168,Z 514.975,A -85,B 0,C 180,E1 -28207.319,E2 -28207.319} C_VEL
LIN {X 0,Y 86.052,Z 508.351,A -85,B 0,C 180,E1 -28212.688,E2 -28212.688} C_VEL
LIN {X 0,Y 88.989,Z 504.245,A -85,B 0,C 180,E1 -28215.31,E2 -28215.31} C_VEL
LIN {X 0,Y 91.865,Z 497.011,A -85,B 0,C 180,E1 -28219.922,E2 -28219.922} C_VEL
LIN {X 0,Y 95.056,Z 487.218,A -85,B 0,C 180,E1 -28225.236,E2 -28225.236} C_VEL
LIN {X 0,Y 96.105,Z 483.104,A -85,B 0,C 180,E1 -28227.26,E2 -28227.26} C_VEL
LIN {X 0,Y 95.927,Z 479.023,A -85,B 0,C 180,E1 -28229.899,E2 -28229.899} C_VEL
LIN {X 0,Y 94.924,Z 472.199,A -85,B 0,C 180,E1 -28234.803,E2 -28234.803} C_VEL
LIN {X 0,Y 93.536,Z 465.552,A -85,B 0,C 180,E1 -28240.128,E2 -28240.128} C_VEL
LIN {X 0,Y 92.647,Z 461.767,A -85,B 0,C 180,E1 -28243.472,E2 -28243.472} C_VEL
LIN {X 0,Y 91.712,Z 458.568,A -85,B 0,C 180,E1 -28246.709,E2 -28246.709} C_VEL
LIN {X 0,Y 90.491,Z 455.147,A -85,B 0,C 180,E1 -28251.064,E2 -28251.064} C_VEL
LIN {X 0,Y 89.66,Z 453.471,A -85,B 0,C 180,E1 -28253.856,E2 -28253.856} C_VEL
LIN {X 0,Y 87.728,Z 448.909,A -85,B 0,C 180,E1 -28264.595,E2 -28264.595} C_VEL
LIN {X 0,Y 86.933,Z 448.8,A -85,B 0,C 180,E1 -28274.036,E2 -28274.036} C_VEL
LIN {X 0,Y 87.222,Z 449.072,A -85,B 0,C 180,E1 -28278.802,E2 -28278.802} C_VEL
LIN {X 0,Y 88.432,Z 452.95,A -85,B 0,C 180,E1 -28289.033,E2 -28289.033} C_VEL
LIN {X 0,Y 88.996,Z 453.469,A -85,B 0,C 180,E1 -28290.881,E2 -28290.881} C_VEL
LIN {X 0,Y 90.947,Z 457.89,A -85,B 0,C 180,E1 -28298.185,E2 -28298.185} C_VEL
LIN {X 0,Y 93.147,Z 463.192,A -85,B 0,C 180,E1 -28304.885,E2 -28304.885} C_VEL
LIN {X 0,Y 95.159,Z 469.002,A -85,B 0,C 180,E1 -28310.872,E2 -28310.872} C_VEL
LIN {X 0,Y 96.829,Z 475.873,A -85,B 0,C 180,E1 -28316.853,E2 -28316.853} C_VEL
LIN {X 0,Y 97.654,Z 480.893,A -85,B 0,C 180,E1 -28320.907,E2 -28320.907} C_VEL
LIN {X 0,Y 97.815,Z 482.871,A -85,B 0,C 180,E1 -28322.386,E2 -28322.386} C_VEL
LIN {X 0,Y 97.572,Z 484.365,A -85,B 0,C 180,E1 -28323.354,E2 -28323.354} C_VEL
LIN {X 0,Y 96.824,Z 486.048,A -85,B 0,C 180,E1 -28324.174,E2 -28324.174} C_VEL
LIN {X 0,Y 90.797,Z 495.328,A -85,B 0,C 180,E1 -28328.666,E2 -28328.666} C_VEL
LIN {X 0,Y 84.794,Z 503.649,A -85,B 0,C 180,E1 -28334.364,E2 -28334.364} C_VEL
LIN {X 0,Y 79.786,Z 510.22,A -85,B 0,C 180,E1 -28340.661,E2 -28340.661} C_VEL
LIN {X 0,Y 77.02,Z 513.065,A -85,B 0,C 180,E1 -28343.865,E2 -28343.865} C_VEL
LIN {X 0,Y 71.223,Z 517.215,A -85,B 0,C 180,E1 -28349.208,E2 -28349.208} C_VEL
LIN {X 0,Y 66.787,Z 520.023,A -85,B 0,C 180,E1 -28354.213,E2 -28354.213} C_VEL
LIN {X 0,Y 64.45,Z 521.846,A -85,B 0,C 180,E1 -28358.722,E2 -28358.722} C_VEL
LIN {X 0,Y 63.992,Z 522.397,A -85,B 0,C 180,E1 -28360.372,E2 -28360.372} C_VEL
LIN {X 0,Y 62.806,Z 524.935,A -85,B 0,C 180,E1 -28369.602,E2 -28369.602} C_VEL
LIN {X 0,Y 62.969,Z 526.28,A -85,B 0,C 180,E1 -28376.763,E2 -28376.763} C_VEL
LIN {X 0,Y 63.788,Z 527.085,A -85,B 0,C 180,E1 -28383.412,E2 -28383.412} C_VEL
LIN {X 0,Y 66.071,Z 527.529,A -85,B 0,C 180,E1 -28391.877,E2 -28391.877} C_VEL
LIN {X 0,Y 71.035,Z 526.905,A -85,B 0,C 180,E1 -28402.306,E2 -28402.306} C_VEL
LIN {X 0,Y 74.813,Z 525.925,A -85,B 0,C 180,E1 -28407.701,E2 -28407.701} C_VEL
LIN {X 0,Y 80.85,Z 523.765,A -85,B 0,C 180,E1 -28414.239,E2 -28414.239} C_VEL
LIN {X 0,Y 89.232,Z 519.913,A -85,B 0,C 180,E1 -28420.902,E2 -28420.902} C_VEL
LIN {X 0,Y 97.796,Z 514.993,A -85,B 0,C 180,E1 -28425.93,E2 -28425.93} C_VEL
LIN {X 0,Y 106.963,Z 508.591,A -85,B 0,C 180,E1 -28430.208,E2 -28430.208} C_VEL
LIN {X 0,Y 108.797,Z 506.971,A -85,B 0,C 180,E1 -28431.477,E2 -28431.477} C_VEL
LIN {X 0,Y 110.042,Z 504.524,A -85,B 0,C 180,E1 -28436.339,E2 -28436.339} C_VEL
LIN {X 0,Y 110.729,Z 503.082,A -85,B 0,C 180,E1 -28440,E2 -28440} C_VEL
LIN {X 0,Y 111.405,Z 501.987,A -85,B 0,C 180,E1 -28443.617,E2 -28443.617} C_VEL
LIN {X 0,Y 111.119,Z 502.002,A -85,B 0,C 180,E1 -28447.267,E2 -28447.267} C_VEL
LIN {X 0,Y 110.717,Z 502.528,A -85,B 0,C 180,E1 -28450.978,E2 -28450.978} C_VEL
LIN {X 0,Y 110.046,Z 504.197,A -85,B 0,C 180,E1 -28456.7,E2 -28456.7} C_VEL
LIN {X 0,Y 109.337,Z 506.043,A -85,B 0,C 180,E1 -28460.704,E2 -28460.704} C_VEL
LIN {X 0,Y 108.218,Z 508.523,A -85,B 0,C 180,E1 -28464.624,E2 -28464.624} C_VEL
LIN {X 0,Y 107.312,Z 510.385,A -85,B 0,C 180,E1 -28467.287,E2 -28467.287} C_VEL
LIN {X 0,Y 104.767,Z 512.993,A -85,B 0,C 180,E1 -28469.318,E2 -28469.318} C_VEL
LIN {X 0,Y 99.97,Z 517.164,A -85,B 0,C 180,E1 -28472.493,E2 -28472.493} C_VEL
LIN {X 0,Y 91.9,Z 522.516,A -85,B 0,C 180,E1 -28476.6,E2 -28476.6} C_VEL
LIN {X 0,Y 82.992,Z 527.551,A -85,B 0,C 180,E1 -28482.646,E2 -28482.646} C_VEL
LIN {X 0,Y 75.757,Z 530.944,A -85,B 0,C 180,E1 -28489.519,E2 -28489.519} C_VEL
LIN {X 0,Y 68.85,Z 533.473,A -85,B 0,C 180,E1 -28499.324,E2 -28499.324} C_VEL
LIN {X 0,Y 64.534,Z 534.539,A -85,B 0,C 180,E1 -28510.944,E2 -28510.944} C_VEL
LIN {X 0,Y 63.428,Z 534.492,A -85,B 0,C 180,E1 -28517.209,E2 -28517.209} C_VEL
LIN {X 0,Y 63.012,Z 534.054,A -85,B 0,C 180,E1 -28523.609,E2 -28523.609} C_VEL
LIN {X 0,Y 63.191,Z 533.23,A -85,B 0,C 180,E1 -28530.012,E2 -28530.012} C_VEL
LIN {X 0,Y 63.074,Z 531.929,A -85,B 0,C 180,E1 -28536.41,E2 -28536.41} C_VEL
LIN {X 0,Y 64.019,Z 529.112,A -85,B 0,C 180,E1 -28545.941,E2 -28545.941} C_VEL
LIN {X 0,Y 66.476,Z 525.238,A -85,B 0,C 180,E1 -28555.029,E2 -28555.029} C_VEL
LIN {X 0,Y 70.43,Z 520.219,A -85,B 0,C 180,E1 -28563.299,E2 -28563.299} C_VEL
LIN {X 0,Y 75.608,Z 513.884,A -85,B 0,C 180,E1 -28570.605,E2 -28570.605} C_VEL
LIN {X 0,Y 80.388,Z 507.819,A -85,B 0,C 180,E1 -28575.62,E2 -28575.62} C_VEL
LIN {X 0,Y 82.96,Z 504.442,A -85,B 0,C 180,E1 -28577.849,E2 -28577.849} C_VEL
LIN {X 0,Y 86.146,Z 497.32,A -85,B 0,C 180,E1 -28582.709,E2 -28582.709} C_VEL
LIN {X 0,Y 89.624,Z 487.914,A -85,B 0,C 180,E1 -28588.126,E2 -28588.126} C_VEL
